# B&R Automation Studio project Parker_BMM_ST_V5_3147_V12 (part 11)

#### extrlift.c
```c
/********************************************************************
 * COPYRIGHT --  B&R China
 ********************************************************************
 * Program: extrlift
 * File: extrlift.c
 * Author: lijianjun
 * Created: March 06, 2013
 ********************************************************************
 * Implementation of program extrlift --- upward and downward
 ********************************************************************/

#include <bur/plctypes.h>

#ifdef _DEFAULT_INCLUDES
#include <AsDefault.h>
#endif

#define   INSTANCY_STOP_DECEL       3000

#define   INSTANCY_STOP_UP_DECEL    3000
#define   INSTANCY_STOP_DN_DECEL    3000
/**************************************************************************************
                            Function Declarations
**************************************************************************************/
void ExtrLiftTime( Mold_typ * pMold);
void ExtrLiftInverter( Mold_typ * pMold);
void ExtrLiftSwitch( Mold_typ * pMold);
void ExtrLiftDriveToggle_Drive(Mold_typ * pMold, ExtrLift_Fix_typ * pExtrLiftFix, ExtrLift_Para_typ * pExtrLiftPara);
REAL xTogLinearRTrans(REAL pTogLinPos);
/**************************************************************************************
     	        		I N I T U P  O F   T H E   T A S K
**************************************************************************************/
_INIT void init ( void )
{
	RTInfo_Task.enable = 1;
	RTInfo(&RTInfo_Task);

	tTask = RTInfo_Task.cycle_time/1000.0/1000.0;		/*  from us ---> s  */

	LMold.ExtrLift.Step = 30000;
	RMold.ExtrLift.Step = 30000;

	RMold.ExtrLift.vProfGen.Ts    = tTask;
	RMold.ExtrLift.vProfGen.accel = 800.0;
	RMold.ExtrLift.vProfGen.decel = 600.0;
	RMold.ExtrLift.vRamp.Ts       = tTask;
	RMold.ExtrLift.vRamp.Accel    = 1000;

	LMold.ExtrLift.vProfGen.Ts    = tTask;
	LMold.ExtrLift.vProfGen.accel = 800.0;
	LMold.ExtrLift.vProfGen.decel = 600.0;
	LMold.ExtrLift.vRamp.Ts       = tTask;
	LMold.ExtrLift.vRamp.Accel    = 1000;

	/* differentiator for evaluating the actual speed */
	vActHydDT2_L.Ts = tTask;	/* cycle time tTasks 			  */
	vActHydDT2_L.Tv = 1.0; 	/* derivative time constant [s]   */
	vActHydDT2_L.T1 = 5 * tTask; 	/* filter time constant 1 : 0.01s */
	vActHydDT2_L.T2 = 5 * tTask; 	/* filter time constant 2 : 0.01s */

	/* differentiator for evaluating the actual speed */
	vActHydDT2_R.Ts = tTask;	/* cycle time tTasks 			  */
	vActHydDT2_R.Tv = 1.0; 	/* derivative time constant [s]   */
	vActHydDT2_R.T1 = 5 * tTask; 	/* filter time constant 1 : 0.01s */
	vActHydDT2_R.T2 = 5 * tTask; 	/* filter time constant 2 : 0.01s */

	if( 10 > gMachineFix.ExtrLift.ToggleLinNodeNum ) gMachineFix.ExtrLift.ToggleLinNodeNum = 10;
	ToggleLinNodeNum = gMachineFix.ExtrLift.ToggleLinNodeNum;
	/* extrlift toggle linear */

	TogLinearR.enable = 1;
	TogLinearR.nNodes = ToggleLinNodeNum;
	TogLinearR.pNodes = &gMachineFix.ExtrLift.ToggleLin[0];

	xTogLinearR.enable = 1;
	xTogLinearR.nNodes = ToggleLinNodeNum;
	xTogLinearR.pNodes = &xToggleNodeR[0];

	memcpy(ToggleROld,gMachineFix.ExtrLift.ToggleLin,sizeof(gMachineFix.ExtrLift.ToggleLin));

} /* end of _INIT */

 /*************************************************************************************
        				C Y C L I C   P A R T   O F   T H E   T A S K
**************************************************************************************/

_CYCLIC void cyclic ( void )
{
	if(gMachinePara.ExtrLiftLower.accel < 20.0)gMachinePara.ExtrLiftLower.accel = 20.0;

	if(1 == gMachineIn.ExtrLiftInverterFault)
	{
		cntTime = cntTime + 1;
		if(cntTime >10000)cntTime =1000;
	}
	else
	{
		cntTime = 0;
	}

	if(cntTime > 100)
	{
		gAlarm.SwingInvertErr = 1;
	}

	/*--- 機構線性，強制線性化 ----*/
	if( ACTUATOR_ELECTRIC ==  gMachineFix.ExtrLift.eActuatorType)
	{
		int ToggleLinIndex;
		if( MECHANISM_LINEAR ==  gMachineFix.ExtrLift.eMechanismType )
		{
			bToggle_Init = 1;
			for(ToggleLinIndex = 1;ToggleLinIndex < (MAX_TOGGLE_LIN_NUM); ToggleLinIndex++)
			{
				int iSumR = 0;
				iSumR = gMachineFix.ExtrLift.Length / (ToggleLinNodeNum);
				gMachineFix.ExtrLift.ToggleLin[ToggleLinIndex].X = iSumR * ToggleLinIndex ;
				gMachineFix.ExtrLift.ToggleLin[ToggleLinIndex].Y = iSumR * ToggleLinIndex ;

				if( ToggleLinIndex >= ToggleLinNodeNum)
				{
					gMachineFix.ExtrLift.ToggleLin[ToggleLinIndex].X = gMachineFix.ExtrLift.Length ;
					gMachineFix.ExtrLift.ToggleLin[ToggleLinIndex].Y = gMachineFix.ExtrLift.Length ;
				}

			}
		}
		else if( MECHANISM_TOGGLE ==  gMachineFix.ExtrLift.eMechanismType  )
		{
			if(1 == bToggle_Init)
			{
				bToggle_Init = 0;

				// clear ToggleLin table
				for(ToggleLinIndex = 1;ToggleLinIndex < (MAX_TOGGLE_LIN_NUM); ToggleLinIndex++)
				{

					if(ToggleLinIndex <ToggleLinNodeNum )
					{
						gMachineFix.ExtrLift.ToggleLin[ToggleLinIndex].X = 0 ;
						gMachineFix.ExtrLift.ToggleLin[ToggleLinIndex].Y = 0 ;
					}
					else
					{
						gMachineFix.ExtrLift.ToggleLin[ToggleLinIndex].X = gMachineFix.ExtrLift.Length ;
						gMachineFix.ExtrLift.ToggleLin[ToggleLinIndex].Y = gMachineFix.ExtrLift.Length ;
					}
				}

			}
		}
	}

	int i;
	for(i=0;i<MAX_TOGGLE_LIN_NUM;i++)
	{
		xToggleNodeR[i].X = gMachineFix.ExtrLift.ToggleLin[i].Y;
		xToggleNodeR[i].Y = gMachineFix.ExtrLift.ToggleLin[i].X;
	}

	if( 10 > gMachineFix.ExtrLift.ToggleLinNodeNum ) gMachineFix.ExtrLift.ToggleLinNodeNum = 10;
	else if( 30 < gMachineFix.ExtrLift.ToggleLinNodeNum ) gMachineFix.ExtrLift.ToggleLinNodeNum = 30;
	ToggleLinNodeNum = gMachineFix.ExtrLift.ToggleLinNodeNum;
	//TogLinear  update

	if(memcmp(ToggleROld,gMachineFix.ExtrLift.ToggleLin,sizeof(gMachineFix.ExtrLift.ToggleLin)) != 0
		|| oldToggleLinNodeNum != ToggleLinNodeNum)
	{
		TogLinearR.update = 1;
		TogLinearR.nNodes = ToggleLinNodeNum;
		memcpy(ToggleROld,gMachineFix.ExtrLift.ToggleLin,sizeof(gMachineFix.ExtrLift.ToggleLin));

		xTogLinearR.update = 1;
		xTogLinearR.nNodes = ToggleLinNodeNum;
		HydLinear(&xTogLinearR);
	}

	oldToggleLinNodeNum = ToggleLinNodeNum;

	/*  ExtruderLift Up & Dn limit   */
	RMold.TransDIn.ExtruderLiftUpLimit = gMachineIn.ExtruderLiftUpLimit;
	LMold.TransDIn.ExtruderLiftUpLimit = gMachineIn.ExtruderLiftUpLimit;

	RMold.TransDIn.ExtruderLiftDnLimit = gMachineIn.ExtruderLiftDnLimit;
	LMold.TransDIn.ExtruderLiftDnLimit = gMachineIn.ExtruderLiftDnLimit;

	/*  valve output*/
	gMachineOut.ExtrLiftUp 		= (LMold.ValveOut.ExtrLiftUp| RMold.ValveOut.ExtrLiftUp);
	gMachineOut.ExtrLiftUpCheck = (LMold.ValveOut.ExtrLiftUpCheck| RMold.ValveOut.ExtrLiftUpCheck);  /* 上止回閥*/
	if(1 == gMachineFix.Option.bExtrLiftUpFastValve)
	{
		gMachineOut.ExtrLiftUpFast  = (LMold.ValveOut.ExtrLiftUpFast | RMold.ValveOut.ExtrLiftUpFast);	 /* 上快速閥*/
	}
	gMachineOut.ExtrLiftDn 		= (LMold.ValveOut.ExtrLiftDn | RMold.ValveOut.ExtrLiftDn);

	/* velocity  */

	if(ACTUATOR_HYD == gMachineFix.ExtrLift.eActuatorType)
	{
		vActHydDT2_R.u = RMold.ExtrLift.mmAs;
	}
	else if(ACTUATOR_ELECTRIC == gMachineFix.ExtrLift.eActuatorType)
	{
		if(TogLinearR.status != 0)  //LinNotOK
		{
			vActHydDT2_R.u = RMold.ExtrLift.mmAs;
		}
		else
		{
			vActHydDT2_R.u = RMold.ExtrLift.mmAsDrive;
		}
	}

	HydDT2(&vActHydDT2_R);
	RMold.ExtrLift.v_act = vActHydDT2_R.y;

	/*  run function  */
	if(ACTUATOR_HYD == gMachineFix.ExtrLift.eActuatorType) //Hydraulic
	{
		if(0 == gMachineFix.Option.bHideLeftStation)  // two mold
		{
			ExtrLiftSwitch(&LMold);
		}
		ExtrLiftSwitch(&RMold);
	}
	else if(ACTUATOR_ELECTRIC == gMachineFix.ExtrLift.eActuatorType) //Electric
	{
		//		if(0 == gMachineFix.Option.bHideLeftStation)  // two mold
		//		{
		//			ExtrLiftDriveToggle_Drive(&LMold, &gMachineFix.ExtrLift, &gMachinePara.Extrlift);
		//		}
		ExtrLiftDriveToggle_Drive(&RMold, &gMachineFix.ExtrLift, &gMachinePara.Extrlift);
	}

	/*------------- ActuatorType--------------- */
	gMachineFix.ExtrLift.eActuatorType;

	/*------------ PressueOutputType--------------- */
	gMachineFix.ExtrLift.ePressueOutputType;

	/*------------ FluxOutputType--------------- */
	gMachineFix.ExtrLift.eFluxOutputType;

	/*---------------Motor Trand-------------*/
	gMotorTrace.Extrlift.Position 		= RMold.ExtrLift.mmAs;

} /* end of _CYCLIC */

void ExtrLiftTime( Mold_typ * pMold)
{

	/* ------------------ Step Machine Control ------------------ */
	switch ( pMold->ExtrLift.Step )
	{
		/*------------------ stop all the output ------------------*/
		case 0:
			pMold->ValveOut.ExtrLiftUp  = 0;
			pMold->ActInfo.ExtrLiftUp = 0;
			pMold->ActInfo.ExtrLiftDn = 0;

			pMold->ExtrLift.Timer.IN = 0;
			break;

		/*------------------ Extr Lift -------------------- */
		case 100: 	/* ExtrLift delay*/

			if(pMold->TimeSet.ExtrLiftUpDelay != 0)
			{
				pMold->ExtrLift.Timer.IN = 1;
				pMold->ExtrLift.Timer.PT = pMold->TimeSet.ExtrLiftUpDelay;
				pMold->ExtrLift.Step 	= 200;
			}
			else
			{
				pMold->ExtrLift.Step = 300;
			}
			break;

		case 200: 	/* delay ok */
			pMold->TimeDis.ExtrLiftUpDelay = pMold->ExtrLift.Timer.ET;
			if (1 == pMold->ExtrLift.Timer.Q)
			{
				pMold->ExtrLift.Timer.IN     = 0;
				//				pMold->TimeDis.ExtrLiftUpDelay = 0;
				pMold->ExtrLift.Step = 300;
			}
			break;

		case 300:
			if(pMold->TimeSet.ExtrLiftUpHoldTime != 0)
			{
				pMold->ExtrLift.Timer.IN = 1;
				pMold->ExtrLift.Timer.PT = pMold->TimeSet.ExtrLiftUpHoldTime;
				pMold->ExtrLift.Step = 400;
			}
			else
			{
				pMold->ExtrLift.Step = 2900;
			}
			break;

		case 400:
			pMold->ActInfo.ExtrLiftUp = 1;
			pMold->ActInfo.ExtrLiftDn = 0;
			pMold->ValveOut.ExtrLiftUp       = 1;

			pMold->TimeDis.ExtrLiftUpHoldTime = pMold->ExtrLift.Timer.ET;
			if (1 == pMold->ExtrLift.Timer.Q)
			{
				pMold->ValveOut.ExtrLiftUp     = 0;
				pMold->ExtrLift.Timer.IN = 0;
				//				pMold->TimeDis.ExtrLiftUpHoldTime = 0;
				pMold->ExtrLift.Step = 500;
			}
			break;

		case 500:
			pMold->ActInfo.ExtrLiftUp = 0;
			pMold->ActInfo.ExtrLiftDn = 0;/*Test*/
			pMold->ValveOut.ExtrLiftUp       = 0;

			pMold->ExtrLift.Step = 2900;
			break;

		case 2900:
			pMold->ExtrLift.Timer.IN    = 0;

			pMold->TimeDis.ExtrLiftUpDelay = 0;
			pMold->TimeDis.ExtrLiftUpHoldTime = 0;
			pMold->TimeDis.ExtrLiftSlowTime = 0;

			pMold->ActInfo.ExtrLiftUp = 0;
			pMold->ActInfo.ExtrLiftDn = 0;
			pMold->ValveOut.ExtrLiftUp       = 0;

			pMold->ExtrLift.Step = 3000;
			break;
		case 3000:
			break;

		case 5000:					/*  Manual up */

			pMold->ActInfo.ExtrLiftUp = 1;
			pMold->ActInfo.ExtrLiftDn = 0;

			if((0 == pMold->TransDIn.ExtruderLiftUpLimit) && (0 == pMold->TransDIn.ExtruderLiftDnLimit))
			{
				pMold->ValveOut.ExtrLiftUp       = 0;
			}
			else
			{
				if(1 == pMold->TransDIn.ExtruderLiftUpLimit)
				{
					pMold->ValveOut.ExtrLiftUp       = 0;
				}
				else
				{
					pMold->ValveOut.ExtrLiftUp       = 1;
				}
			}
			break;

		case 15000:					/*  Manual down */
			pMold->ActInfo.ExtrLiftUp = 0;
			pMold->ActInfo.ExtrLiftDn = 0;
			pMold->ValveOut.ExtrLiftUp       = 0;

			break;

		/*--------------- Manual action stop -----------------*/
		case 20000:
			pMold->ExtrLift.Timer.IN = 0;

			pMold->ActInfo.ExtrLiftUp = 0;
			pMold->ActInfo.ExtrLiftDn = 0;
			pMold->ValveOut.ExtrLiftUp       = 0;

			pMold->ExtrLift.Step = 0;
			break;

		/*--------------- Instance stop -----------------*/
		case 30000:
			pMold->ExtrLift.Timer.IN = 0;

			pMold->ActInfo.ExtrLiftUp = 0;
			pMold->ActInfo.ExtrLiftDn = 0;
			pMold->ValveOut.ExtrLiftUp       = 0;

			pMold->ExtrLift.Step = 0;
			break;

		/*--------------- error -----------------*/
		case 40000:
			pMold->ExtrLift.Timer.IN  = 0;
			pMold->ActInfo.ExtrLiftUp = 0;
			pMold->ActInfo.ExtrLiftDn = 0;
			pMold->ValveOut.ExtrLiftUp       = 0;

			pMold->ExtrLift.Step = 0;
			break;
	}/* end of switch */
}/*end of function */

void ExtrLiftInverter( Mold_typ * pMold)
{
	if(0 == pMold->TimeSet.ExtrLiftSlowTime)pMold->TimeSet.ExtrLiftSlowTime = 1000;

	switch ( pMold->ExtrLift.Step)
	{
		/*------------------ stop all the output ------------------*/
		case 0:
			pMold->ValveOut.ExtrLiftUp   = 0;
			pMold->ExtrLift.v_set = 0.0;

			pMold->ActInfo.ExtrLiftUp = 0;
			pMold->ActInfo.ExtrLiftDn = 0;

			pMold->ExtrLift.Timer.IN = 0;
			break;

		/*------------------ Extr Lift -------------------- */
		case 100: 	/* ExtrLift delay*/
			if(pMold->TimeSet.ExtrLiftUpDelay != 0)
			{
				pMold->ExtrLift.Timer.IN = 1;
				pMold->ExtrLift.Timer.PT = pMold->TimeSet.ExtrLiftUpDelay;
				pMold->ExtrLift.Step 	= 200;
			}
			else
			{
				pMold->ExtrLift.Step = 300;
			}
			break;

		case 200: 	/* delay ok */
			pMold->TimeDis.ExtrLiftUpDelay = pMold->ExtrLift.Timer.ET;
			if (1 == pMold->ExtrLift.Timer.Q)
			{
				pMold->ExtrLift.Timer.IN     = 0;
				pMold->TimeDis.ExtrLiftUpDelay = 0;
				pMold->ExtrLift.Step = 300;
			}
			break;

		case 300:
			pMold->ExtrLift.Timer.IN = 1;
			pMold->ExtrLift.Timer.PT = pMold->TimeSet.ExtrLiftSlowTime;

			pMold->ExtrLift.vRamp.Internal.Once = 0;
			pMold->ExtrLift.vRamp.Set = 0.0;

			pMold->ExtrLift.vRamp.Ts = 0.002;
			pMold->ExtrLift.vRamp.Accel = gMachinePara.ExtrLiftLower.accel;
			if(pMold->ExtrLift.vRamp.Accel < 10)pMold->ExtrLift.vRamp.Accel = 100;

			HydSCurveRamp(&pMold->ExtrLift.vRamp);
			pMold->ExtrLift.v_set = pMold->ExtrLift.vRamp.Out;

			pMold->ExtrLift.Step = 400;
			break;

		case 400:
			pMold->ActInfo.ExtrLiftUp = 1;
			pMold->ActInfo.ExtrLiftDn = 0;
			pMold->ValveOut.ExtrLiftUp       = 1;

			pMold->ExtrLift.vRamp.Set = gMachinePara.ExtrLiftLower.vLowerQuick;
			HydSCurveRamp(&pMold->ExtrLift.vRamp);
			pMold->ExtrLift.v_set = pMold->ExtrLift.vRamp.Out;

			pMold->TimeDis.ExtrLiftUpHoldTime = pMold->ExtrLift.Timer.ET;
			if(1 == gMachineIn.ExtrLowerSlowLimit || pMold->TimeDis.ExtrLiftUpHoldTime >= pMold->TimeSet.ExtrLiftUpHoldTime )
			{
				pMold->ExtrLift.Step = 500;
			}

			pMold->TimeDis.ExtrLiftSlowTime = pMold->ExtrLift.Timer.ET;
			if (1 == pMold->ExtrLift.Timer.Q)
			{
				pMold->ExtrLift.v_set = 0.0;
				pMold->ValveOut.ExtrLiftUp      = 0;
				pMold->ExtrLift.Timer.IN = 0;
				pMold->ExtrLift.Step = 40000;
			}
			break;

		case 500:
			pMold->ValveOut.ExtrLiftUp = 1;

			pMold->ExtrLift.vRamp.Set = gMachinePara.ExtrLiftLower.vLowerSlow;
			HydSCurveRamp(&pMold->ExtrLift.vRamp);
			pMold->ExtrLift.v_set = pMold->ExtrLift.vRamp.Out;

			pMold->TimeDis.ExtrLiftSlowTime = pMold->ExtrLift.Timer.ET;
			if (1 == pMold->ExtrLift.Timer.Q)
			{
				pMold->ExtrLift.v_set = 0.0;
				pMold->ValveOut.ExtrLiftUp      = 0;
				pMold->ExtrLift.Timer.IN = 0;
				pMold->ExtrLift.Step = 40000;
			}

			if(1 == gMachineIn.ExtrLowerLimit)
			{
				pMold->ExtrLift.Timer.IN = 0;
				pMold->ExtrLift.Step = 600;
			}
			break;

		case 600:
			pMold->ExtrLift.vRamp.Accel = 1600;
			pMold->ExtrLift.vRamp.Set = 0.0;
			HydSCurveRamp(&pMold->ExtrLift.vRamp);
			pMold->ExtrLift.v_set = pMold->ExtrLift.vRamp.Out;

			if(pMold->ExtrLift.v_set < 0.1 && pMold->ExtrLift.v_set > -0.1)
			{
				pMold->ExtrLift.v_set = 0.0;
				pMold->ExtrLift.Step = 700;
			}
			break;

		case 700:
			pMold->ActInfo.ExtrLiftUp = 0;
			pMold->ActInfo.ExtrLiftDn = 0;
			pMold->ValveOut.ExtrLiftUp       = 0;
			pMold->ExtrLift.v_set     = 0.0;

			pMold->ExtrLift.Step = 2900;
			break;

		case 2900:
			pMold->ExtrLift.Timer.IN    = 0;

			pMold->TimeDis.ExtrLiftUpDelay = 0;

			pMold->ActInfo.ExtrLiftUp = 0;
			pMold->ActInfo.ExtrLiftDn = 0;
			pMold->ValveOut.ExtrLiftUp       = 0;
			pMold->ExtrLift.v_set     = 0.0;

			pMold->ExtrLift.Step = 3000;
			break;
		case 3000:
			break;

		case 5000:					/*  Manual up */
			pMold->ActInfo.ExtrLiftUp = 1;
			pMold->ActInfo.ExtrLiftDn = 0;
			pMold->ValveOut.ExtrLiftUp       = 1;

			pMold->ExtrLift.v_set = gMachinePara.ExtrLiftLower.vLowerSlow;
			break;

		case 15000:					/*  Manual down */
			pMold->ActInfo.ExtrLiftUp = 0;
			pMold->ActInfo.ExtrLiftDn = 0;
			pMold->ValveOut.ExtrLiftUp       = 0;
			break;

		/*--------------- Manual action stop -----------------*/
		case 20000:
			pMold->ExtrLift.Timer.IN = 0;

			pMold->ActInfo.ExtrLiftUp = 0;
			pMold->ActInfo.ExtrLiftDn = 0;
			pMold->ValveOut.ExtrLiftUp       = 0;

			pMold->ExtrLift.vRamp.Internal.Once = 0;
			pMold->ExtrLift.vRamp.Set = pMold->ExtrLift.v_set;

			pMold->ExtrLift.vRamp.Ts = 0.002;
			pMold->ExtrLift.vRamp.Accel = gMachinePara.ExtrLiftLower.accel;
			if(pMold->ExtrLift.vRamp.Accel < 10)pMold->ExtrLift.vRamp.Accel = 100;

			HydSCurveRamp(&pMold->ExtrLift.vRamp);
			pMold->ExtrLift.v_set = pMold->ExtrLift.vRamp.Out;

			pMold->ExtrLift.Step = 21000;
			break;

		case 21000:
			pMold->ExtrLift.vRamp.Accel = 2000;
			pMold->ExtrLift.vRamp.Set = 0.0;
			HydSCurveRamp(&pMold->ExtrLift.vRamp);
			pMold->ExtrLift.v_set = pMold->ExtrLift.vRamp.Out;

			if(pMold->ExtrLift.v_set < 0.1 && pMold->ExtrLift.v_set > -0.1)
			{
				pMold->ExtrLift.v_set = 0.0;
				pMold->ExtrLift.Step = 0;
			}
			break;

		/*--------------- Instance stop -----------------*/
		case 30000:
			pMold->ExtrLift.Timer.IN = 0;

			pMold->ActInfo.ExtrLiftUp = 0;
			pMold->ActInfo.ExtrLiftDn = 0;
			pMold->ValveOut.ExtrLiftUp   = 0;
			pMold->ExtrLift.v_set = 0.0;

			pMold->ExtrLift.Step = 0;
			break;

		/*--------------- error -----------------*/
		case 40000:
			pMold->ExtrLift.Timer.IN  = 0;
			pMold->ActInfo.ExtrLiftUp = 0;
			pMold->ActInfo.ExtrLiftDn = 0;
			pMold->ValveOut.ExtrLiftUp   = 0;
			pMold->ExtrLift.v_set = 0.0;

			pMold->ExtrLift.Step = 0;
			break;
	}/* end of switch */

}/*end of function */

void ExtrLiftSwitch( Mold_typ * pMold)
{
	switch ( pMold->ExtrLift.Step )
	{
		/*------------------ stop all the output ------------------*/
		case 0:
			pMold->ActInfo.ExtrLiftUp = 0;
			pMold->ActInfo.ExtrLiftDn = 0;
			pMold->ValveOut.ExtrLiftUp     = 0;
			pMold->ValveOut.ExtrLiftUpCheck    = 0;
			pMold->ValveOut.ExtrLiftUpFast     = 0;
			pMold->ValveOut.ExtrLiftDn 	 = 0;

			pMold->ExtrLift.Timer.IN = 0;
			pMold->ExtrLift.LimitTimer.IN = 0; //ipis0219
			break;

		/*------------------ Extr Lift up-------------------- */
		case 100: 	/* ExtrLift delay*/
			if(pMold->Option.ExtrLift)
			{
				if(pMold->TimeSet.ExtrLiftUpDelay != 0)
				{
					pMold->ExtrLift.Timer.IN = 1;
					pMold->ExtrLift.Timer.PT = pMold->TimeSet.ExtrLiftUpDelay;
					pMold->ExtrLift.Step 	= 200;
				}
				else
				{
					pMold->ExtrLift.Step = 300;
				}
			}
			else
			{
				pMold->ExtrLift.Step = 2900;
			}
			break;

		case 200: 	/* delay ok */
			pMold->TimeDis.ExtrLiftUpDelay = pMold->ExtrLift.Timer.ET;
			if (1 == pMold->ExtrLift.Timer.Q)
			{
				pMold->ExtrLift.Timer.IN     = 0;
				//	pMold->TimeDis.ExtrLiftUpDelay = 0;

				pMold->ExtrLift.Step = 300;
			}
			break;

		case 300:
			if (0 == pMold->TransDIn.ExtruderLiftUpLimit)
			{
				pMold->ExtrLift.LimitTimer.IN = 1; //ipis0219
				pMold->ExtrLift.LimitTimer.PT = pMold->TimeSet.ExtrLiftUpAlarmTime; //ipis0219

				pMold->ExtrLift.Step = 400;
			}
			else
			{
				pMold->ExtrLift.Step = 500;
			}
			break;

		case 400:
			pMold->ActInfo.ExtrLiftUp = 1;
			pMold->ActInfo.ExtrLiftDn = 0;
			pMold->ValveOut.ExtrLiftUp   = 1;
			pMold->ValveOut.ExtrLiftUpCheck    = 0;
			pMold->ValveOut.ExtrLiftUpFast     = 1;
			pMold->ValveOut.ExtrLiftDn 	 = 0;

			pMold->TimeDis.ExtrLiftUpAlarmTime = pMold->ExtrLift.LimitTimer.ET;

			if (1 == pMold->TransDIn.ExtruderLiftUpLimit)
			{

				if(pMold->TimeSet.ExtrLiftUpHoldTime != 0)
				{
					pMold->ExtrLift.Timer.IN = 1;
					pMold->ExtrLift.Timer.PT = pMold->TimeSet.ExtrLiftUpHoldTime;
					pMold->ExtrLift.Step = 450;
				}
				else
				{
					pMold->ExtrLift.Step = 500;
				}
			}
			break;
		case 450:
			pMold->ValveOut.ExtrLiftUpFast     = 0;

			pMold->TimeDis.ExtrLiftUpHoldTime = pMold->ExtrLift.Timer.ET;
			if (1 == pMold->ExtrLift.Timer.Q)
			{
				pMold->ValveOut.ExtrLiftUp      = 0;
				pMold->ExtrLift.Timer.IN = 0;

				pMold->ExtrLift.Step = 500;
			}

			break;

		case 500:
			pMold->ActInfo.ExtrLiftUp = 0;
			pMold->ActInfo.ExtrLiftDn = 0;
			pMold->ValveOut.ExtrLiftUp      = 0;
			pMold->ValveOut.ExtrLiftUpCheck    = 0;
			pMold->ValveOut.ExtrLiftUpFast     = 0;
			pMold->ValveOut.ExtrLiftDn 	  = 0;

			pMold->ExtrLift.LimitTimer.IN = 0;
			if (1 == gMachineInfo.Auto)
			{
				pMold->ExtrLift.Step = 10100;
			}
			else
			{
				pMold->ExtrLift.Step = 2900;
			}

			break;

		case 2900:
			pMold->ExtrLift.Timer.IN    = 0;
			pMold->ExtrLift.LimitTimer.IN = 0;

			//			//gExSPC
			//			if(pMold == & LMold)
			//			{
			//				gExSPC[ExIndex].LMold.tExtrLift = pMold->ExtrLift.LimitTimer.ET/100.0;
			//			}
			//			else
			//			{
			//				gExSPC[ExIndex].RMold.tExtrLift = pMold->ExtrLift.LimitTimer.ET/100.0;
			//			}

			//	pMold->TimeDis.ExtrLiftUpDelay = 0;
			//	pMold->TimeDis.ExtrLiftUpHoldTime = 0;
			//	pMold->TimeDis.ExtrLiftDnHoldTime = 0;

			//	pMold->TimeDis.ExtrLiftUpHoldTime = 0;
			//	pMold->TimeDis.ExtrLiftDnHoldTime = 0;

			pMold->ActInfo.ExtrLiftUp = 0;
			pMold->ActInfo.ExtrLiftDn = 0;
			pMold->ValveOut.ExtrLiftUp      = 0;
			pMold->ValveOut.ExtrLiftUpCheck = 0;
			pMold->ValveOut.ExtrLiftUpFast  = 0;
			pMold->ValveOut.ExtrLiftDn 	  = 0;

			pMold->ExtrLift.Step = 3000;
			break;

		case 3000:
			break;

		case 5000:					/*  Manual up */
			pMold->ActInfo.ExtrLiftUp = 1;
			pMold->ActInfo.ExtrLiftDn = 0;

			pMold->ValveOut.ExtrLiftUp    = 1;
			pMold->ValveOut.ExtrLiftUpCheck  = 0;
			pMold->ValveOut.ExtrLiftUpFast   = 0;
			pMold->ValveOut.ExtrLiftDn 	  = 0;

			break;

		/*------------------ Extr Lift down -------------------- */
		case 10100:
			if (pMold->TimeSet.ExtrLiftDnDelay != 0)
			{
				pMold->ExtrLift.Timer.IN = 1;
				pMold->ExtrLift.Timer.PT = pMold->TimeSet.ExtrLiftDnDelay;
				pMold->ExtrLift.Step = 10200;
			}
			else
			{
				pMold->ExtrLift.Step = 10300;
			}
			break;
		case 10200:
			pMold->TimeDis.ExtrLiftDnDelay = pMold->ExtrLift.Timer.ET;
			if (1 == pMold->ExtrLift.Timer.Q)
			{
				pMold->ExtrLift.Timer.IN = 0;
				//	pMold->TimeDis.ExtrLiftDnDelay = 0;
				pMold->ExtrLift.Step = 10300;
			}
			break;
		case 10300:
			if ( 0 == gMachineIn.ExtruderLiftDnLimit)
			{
				pMold->ExtrLift.LimitTimer.IN = 1;
				pMold->ExtrLift.LimitTimer.PT = pMold->TimeSet.ExtrLiftDnAlarmTime;

				pMold->ExtrLift.Step = 10400;
			}
			else
			{
				pMold->ExtrLift.Step = 10500;
			}
			break;
		case 10400:
			pMold->ActInfo.ExtrLiftUp = 0;
			pMold->ActInfo.ExtrLiftDn = 1;
			pMold->ValveOut.ExtrLiftUp  	= 0;
			pMold->ValveOut.ExtrLiftUpCheck = 1;
			pMold->ValveOut.ExtrLiftUpFast  = 0;
			pMold->ValveOut.ExtrLiftDn 	    = 1;

			pMold->TimeDis.ExtrLiftDnAlarmTime = pMold->ExtrLift.LimitTimer.ET;

			if ( 1 == gMachineIn.ExtruderLiftDnLimit)
			{
				if(pMold->TimeSet.ExtrLiftDnHoldTime != 0)
				{
					pMold->ExtrLift.Timer.IN = 1;
					pMold->ExtrLift.Timer.PT = pMold->TimeSet.ExtrLiftDnHoldTime;
					pMold->ExtrLift.Step = 10450;
				}
				else
				{
					pMold->ExtrLift.Step = 10500;
				}
			}
			break;
		case 10450:
			pMold->TimeDis.ExtrLiftDnHoldTime = pMold->ExtrLift.Timer.ET;
			if (1 == pMold->ExtrLift.Timer.Q)
			{
				pMold->ValveOut.ExtrLiftUp    = 0;
				pMold->ValveOut.ExtrLiftUpCheck = 0;
				pMold->ValveOut.ExtrLiftUpFast  = 0;
				pMold->ValveOut.ExtrLiftDn 	  = 0;
				pMold->ExtrLift.Timer.IN = 0;
				//				pMold->TimeDis.ExtrLiftDnHoldTime = 0;
				pMold->ExtrLift.Step = 10500;
			}
			break;
		case 10500:
			pMold->ActInfo.ExtrLiftUp = 0;
			pMold->ActInfo.ExtrLiftDn = 0;
			pMold->ValveOut.ExtrLiftUp      = 0;
			pMold->ValveOut.ExtrLiftUpCheck = 0;
			pMold->ValveOut.ExtrLiftUpFast  = 0;
			pMold->ValveOut.ExtrLiftDn 	  = 0;
			pMold->ExtrLift.Timer.IN    = 0;
			pMold->ExtrLift.LimitTimer.IN = 0;

			pMold->ExtrLift.Step 	  = 13000;
			break;

		case 13000:

			break;

		case 15000:					/*  Manual down */
			pMold->ActInfo.ExtrLiftUp = 0;
			pMold->ActInfo.ExtrLiftDn = 1;
			pMold->ValveOut.ExtrLiftUp    = 0;
			pMold->ValveOut.ExtrLiftUpCheck  = 1;
			pMold->ValveOut.ExtrLiftUpFast   = 0;
			pMold->ValveOut.ExtrLiftDn 	  = 1;

			break;

		/*--------------- Manual action stop -----------------*/
		case 20000:
			pMold->ExtrLift.Timer.IN = 0;

			pMold->ActInfo.ExtrLiftUp = 0;
			pMold->ActInfo.ExtrLiftDn = 0;
			pMold->ValveOut.ExtrLiftUp       = 0;
			pMold->ValveOut.ExtrLiftUpFast 	 = 0;

			pMold->ValveOut.ExtrLiftUpCheck = 0;
			pMold->ValveOut.ExtrLiftDn 	  	= 0;

			pMold->ExtrLift.Step = 0;
			break;

		/*--------------- Instance stop -----------------*/
		case 30000:
			pMold->ExtrLift.Timer.IN = 0;

			pMold->ActInfo.ExtrLiftUp = 0;
			pMold->ActInfo.ExtrLiftDn = 0;
			pMold->ValveOut.ExtrLiftUp       = 0;
			pMold->ValveOut.ExtrLiftUpFast 	 = 0;

			pMold->ValveOut.ExtrLiftUpCheck = 0;
			pMold->ValveOut.ExtrLiftDn 	  	= 0;

			pMold->ExtrLift.Step = 0;
			break;

		/*--------------- error -----------------*/
		case 40000:
			pMold->ExtrLift.Timer.IN  = 0;

			pMold->ActInfo.ExtrLiftUp = 0;
			pMold->ActInfo.ExtrLiftDn = 0;
			pMold->ValveOut.ExtrLiftUp       = 0;
			pMold->ValveOut.ExtrLiftUpFast 	 = 0;

			pMold->ValveOut.ExtrLiftUpCheck = 0;
			pMold->ValveOut.ExtrLiftDn 	  	= 0;

			pMold->ExtrLift.Step = 0;
			break;
	}/* end of switch */

	/* ----------------- ExtrLift Up / down timeout --------------------  */
	if(1 == pMold->ExtrLift.LimitTimer.Q && 1 == gMachineInfo.TimeLimit)
	{
		if(pMold->ExtrLift.Step < 500 && pMold->ExtrLift.Step > 200)		/* ExtrLift Up  */
		{
			pMold->Alarm.ExtrLiftNotAtUpPos = 1;
		}

		if(pMold->ExtrLift.Step < 10500 && pMold->ExtrLift.Step > 10200)		/* ExtrLift Dn  */
		{
			pMold->Alarm.ExtrLiftNotAtDnPos = 1;
		}

		pMold->ExtrLift.LimitTimer.IN = 0;
		pMold->ExtrLift.Step = 40000;

		if(gMachineInfo.Auto)
		{
			gMachineInfo.ExtrliftAlarmReqSemiAutoFlag = 1;
		}
	}
}

void ExtrLiftDriveToggle_Drive(Mold_typ * pMold, ExtrLift_Fix_typ * pExtrLiftFix, ExtrLift_Para_typ * pExtrLiftPara)
{
	if(pMold == & LMold)
	{
		pExtrLiftFix->pMax = 100;
	}
	else
	{
		pExtrLiftFix->pMax = 100;
	}

	if(1 == gMachineOut.OilPump)
	{
		if(tErrorDelay >= tTask)tErrorDelay = tErrorDelay - tTask;
		if(tErrorDelay < tTask)
		{
			if(pMold == & LMold)
			{
				LMold.HwAlarm.ExtrLiftNetworkErr = !LMold.ExtrLift.NetworkInit;
				LMold.HwAlarm.ExtrLiftPowerOn    = !LMold.ExtrLift.PowerOn;
			}
			else
			{
				RMold.HwAlarm.ExtrLiftNetworkErr = !RMold.ExtrLift.NetworkInit;
				RMold.HwAlarm.ExtrLiftPowerOn    = !RMold.ExtrLift.PowerOn;
			}
		}

		if((RMold.HwAlarm.ExtrLiftNetworkErr ||RMold.HwAlarm.ExtrLiftPowerOn)/*||(LMold.HwAlarm.ExtrLiftNetworkErr ||LMold.HwAlarm.ExtrLiftPowerOn)*/)
		{
			gMachineOut.OilPump = 0;
			gPROCESS_info.oilpumpStop = 1;   //request manual mode
		}
	}
	else
	{
		tErrorDelay = 0.5;
		//		if(pMold == & LMold)
		//		{
		////			LMold.HwAlarm.ExtrLiftNetworkErr = 0;
		////			LMold.HwAlarm.ExtrLiftPowerOn    = 0;
		//		}
		//		else
		//		{
		////			RMold.HwAlarm.ExtrLiftNetworkErr = 0;
		////			RMold.HwAlarm.ExtrLiftPowerOn    = 0;
		//		}
	}

	/* ------------- extrLift axis alarms ------------- */

	pMold->HwAlarm.ExtrLiftAxisErr    = RMold.ExtrLift.Error;

	 /*********************************************************************************
  	**                            HMI data value to PLC                             **
  	*********************************************************************************/
	if(pExtrLiftFix->Length < 10.0)pExtrLiftFix->Length = 60.0;
	if(pExtrLiftFix->Tolerance < 0.1)pExtrLiftFix->Tolerance = 2.0;
	pMold->ExtrLift.Tolerance = pExtrLiftFix->Tolerance;

	if(pExtrLiftFix->Up.V_Max < 30.0)pExtrLiftFix->Up.V_Max = 1000.0;
	if(pExtrLiftFix->Dn.V_Max < 30.0)pExtrLiftFix->Dn.V_Max = 1000.0;

	if(pExtrLiftFix->Up.VoltageMax > -3.0)pExtrLiftFix->Up.VoltageMax = -10.0;
	if(pExtrLiftFix->Dn.VoltageMax < 3.0 )pExtrLiftFix->Dn.VoltageMax = 10.0;

	pMold->ExtrLift.S_Up = pExtrLiftPara->S_Up;
	pMold->ExtrLift.V_Up = pExtrLiftPara->V_Up * pExtrLiftFix->Up.V_Max/100.0;

	pMold->ExtrLift.S_Dn = pExtrLiftPara->S_Dn;
	pMold->ExtrLift.V_Dn = pExtrLiftPara->V_Dn * pExtrLiftFix->Dn.V_Max/100.0;

	if(0 == pExtrLiftPara->V_DnReset)pExtrLiftPara->V_DnReset = 2.0;
	pMold->ExtrLift.V_DnReset = pExtrLiftPara->V_DnReset * pExtrLiftFix->Dn.V_Max/100.0;

	if(pExtrLiftFix->Up.accel_stop < 100)pExtrLiftFix->Up.accel_stop = INSTANCY_STOP_UP_DECEL;
	if(pExtrLiftFix->Dn.accel_stop < 100)pExtrLiftFix->Dn.accel_stop = INSTANCY_STOP_DN_DECEL;
    /*********************************************************************************
   **                            linear calibration status                        **
   *********************************************************************************/
   /* get calibration data  */
	if(pExtrLiftFix->Max < pExtrLiftFix->Zero)
	{
		pMold->ExtrLift.ZeroPos = pExtrLiftFix->Max;
		pMold->ExtrLift.MaxPos  = pExtrLiftFix->Zero;
	}
	else
	{
		pMold->ExtrLift.MaxPos  = pExtrLiftFix->Max;
		pMold->ExtrLift.ZeroPos = pExtrLiftFix->Zero;
	}

	if(pMold->ExtrLift.ZeroPos != 0            						&&
		pMold->ExtrLift.MaxPos > (pMold->ExtrLift.ZeroPos + 3000)  	&&
		pMold->ExtrLift.As     > (pMold->ExtrLift.ZeroPos - 1000)   &&
		pMold->ExtrLift.As     < (RMold.ExtrLift.MaxPos  + 5000))
	{
		pMold->ExtrLift.CalOK = pMold->ExtrLift.NetworkInit;
	}
	else
	{
		pMold->ExtrLift.CalOK = 0;
	}

	pExtrLiftFix->CalibOK = pMold->ExtrLift.CalOK;

	if(1 == pMold->ExtrLift.CalOK)
	{
		if(pExtrLiftFix->Max < pExtrLiftFix->Zero)
		{
			pMold->ExtrLift.mmAsDrive = 1.0 *(pMold->ExtrLift.MaxPos - pMold->ExtrLift.As) * pExtrLiftFix->Length /
				(pMold->ExtrLift.MaxPos - pMold->ExtrLift.ZeroPos);
		}
		else
		{
			pMold->ExtrLift.mmAsDrive = 1.0 *(pMold->ExtrLift.As - pMold->ExtrLift.ZeroPos) * pExtrLiftFix->Length /
				(pMold->ExtrLift.MaxPos - pMold->ExtrLift.ZeroPos);
		}
	}
	else
	{
		pMold->ExtrLift.mmAsDrive = pMold->ExtrLift.mmAsDrive;
		//		pMold->ExtrLift.mmAs = pMold->ExtrLift.mmAs;
		if(0 == gMachineInfo.Calib)	/* 非调校模式  */
		{
			if(pMold->ExtrLift.Step > 0 && pMold->ExtrLift.Step < 20000)
			{
				pMold->ExtrLift.Step = 0;
				//	pMold->ExtrLift.Step = 40000; //ipis081
				pMold->Alarm.ExtrliftCalErr = 1;
			}
		}
		else if(0 == pMold->ExtrLift.NetworkInit)
		{
			if(pMold->ExtrLift.Step > 0 && pMold->ExtrLift.Step < 20000)
			{
				pMold->ExtrLift.Step = 0;
			}
		}
	}/* if(1 == pMold->ExtrLift.CalOK) */

	/*  toggle carriage linear  */
	pExtrLiftFix->ToggleLin[0].X = 0.0;
	pExtrLiftFix->ToggleLin[0].Y = 0.0;

	pExtrLiftFix->ToggleLin[ToggleLinNodeNum-1].X = pExtrLiftFix->Length;
	pExtrLiftFix->ToggleLin[ToggleLinNodeNum-1].Y = pExtrLiftFix->Length;

	TogLinearR.Y = pMold->ExtrLift.mmAsDrive;
	HydLinear(&TogLinearR);

	if(TogLinearR.status != 0)
	{
		pMold->Alarm.ExtrliftLinNotOK = 1;
		pMold->ExtrLift.mmAs = pMold->ExtrLift.mmAsDrive;
	}
	else
	{
		pMold->ExtrLift.mmAs = TogLinearR.X;
	}

	/* network and calibration is ok, axis has an error   */
	if(0 == pMold->ExtrLift.AxisReady)
	{
		if(pMold->ExtrLift.Step > 0 && pMold->ExtrLift.Step < 20000)
		{
			pMold->ExtrLift.Step = 30000;
		}
	}

	/*  relative position  */
	pMold->ExtrLift.Ss = pMold->ExtrLift.As;
	pMold->ExtrLift.mmAsMax = pExtrLiftFix->Length + 10;

	/* gAlarm time value    */
	if(!pMold->TimeSet.ExtrLiftUpAlarmTime)pMold->TimeSet.ExtrLiftUpAlarmTime = 1000;   /* 10s  */
	if(!pMold->TimeSet.ExtrLiftDnAlarmTime)pMold->TimeSet.ExtrLiftDnAlarmTime = 1000;   /* 10s  */

	/* Up or down  position flag  */
	if(1 == pMold->ExtrLift.CalOK)
	{
		pMold->ExtrLift.UpPos = pMold->TransDIn.ExtruderLiftUpLimit
			&& (pMold->ExtrLift.mmAs > (pExtrLiftPara->S_Up - pMold->ExtrLift.Tolerance))
			&& (pMold->ExtrLift.mmAs < (pExtrLiftPara->S_Up + pMold->ExtrLift.Tolerance));

		pMold->ExtrLift.DnPos = pMold->TransDIn.ExtruderLiftDnLimit
			&& (pMold->ExtrLift.mmAs < (pExtrLiftPara->S_Dn + pMold->ExtrLift.Tolerance))
			&& (pMold->ExtrLift.mmAs > (pExtrLiftPara->S_Dn - pMold->ExtrLift.Tolerance));

	}
	else
	{
		pMold->ExtrLift.UpPos = 0;
		pMold->ExtrLift.DnPos = 0;
	}

	/* ------------------ current position ------------------ */
	pMold->ExtrLift.vProfGen.s_act = pMold->ExtrLift.mmAsDrive;
	pMold->ExtrLift.vProfGen.v_act = pMold->ExtrLift.v_act;

	/* Up or down move step */
	switch (pMold->ExtrLift.Step )
	{
		/*------------------ stop all the Output ------------------*/
		case 0:

			pMold->ActInfo.ExtrLiftUp  = 0;
			pMold->ActInfo.ExtrLiftDn  = 0;

			pMold->ExtrLift.p_set = 0;
			pMold->ExtrLift.v_set = 0;

			pMold->ExtrLift.Timer.IN = 0;
			pMold->ExtrLift.LimitTimer.IN = 0;
			break;

		/*------------------ Extrlift up -------------------- */
		case 100: /* up delay*/
			if(pMold->Option.ExtrLift)
			{
				if(pMold->TimeSet.ExtrLiftUpDelay != 0)
				{
					pMold->ExtrLift.Timer.IN = 1;
					pMold->ExtrLift.Timer.PT = pMold->TimeSet.ExtrLiftUpDelay;
					pMold->ExtrLift.Step 	= 200;
				}
				else
				{
					pMold->ExtrLift.Step = 300;
				}
			}
			else
			{
				pMold->ExtrLift.Step = 2900;
			}
			break;

		case 200: /*delay ok*/
			pMold->TimeDis.ExtrLiftUpDelay = pMold->ExtrLift.Timer.ET;
			if (1 == pMold->ExtrLift.Timer.Q)
			{
				pMold->ExtrLift.Timer.IN     = 0;
				//	pMold->TimeDis.ExtrLiftUpDelay = 0;
				pMold->ExtrLift.Step = 300;
			}
			break;

		case 300:
			if(0 == pMold->ExtrLift.UpHWSwitch)
			{

				/* xTogLinearLTrans */
				pMold->ExtrLift.S_UpDrive = xTogLinearRTrans(pExtrLiftPara->S_Up);

				pMold->ExtrLift.LimitTimer.IN = 1;
				pMold->ExtrLift.LimitTimer.PT = pMold->TimeSet.ExtrLiftUpAlarmTime;

				pMold->ExtrLift.vProfGen.Ts = tTask;
				pMold->ExtrLift.vProfGen.Tj = pExtrLiftFix->Up.Tj;
				pMold->ExtrLift.vProfGen.Td = pExtrLiftFix->Up.Td;

				pMold->ExtrLift.vProfGen.accel = pExtrLiftFix->Up.accel;
				if(pMold->ExtrLift.vProfGen.accel <= 0.0)pMold->ExtrLift.vProfGen.accel = 1000;

				pMold->ExtrLift.vProfGen.decel = pExtrLiftFix->Up.accel;
				if(pMold->ExtrLift.vProfGen.decel <= 0.0)pMold->ExtrLift.vProfGen.decel = 1000;

				pMold->ExtrLift.vProfGen.decel_end = pExtrLiftFix->Up.decel_end;
				if(pMold->ExtrLift.vProfGen.decel_end <= 0.0)pMold->ExtrLift.vProfGen.decel_end = 100;

				pMold->ExtrLift.vProfGen.v_start = 0;
				pMold->ExtrLift.vProfGen.v_end = 0.0;
				pMold->ExtrLift.vProfGen.s_end = pMold->ExtrLift.S_UpDrive;
				pMold->ExtrLift.vProfGen.init = 1;

				pMold->ExtrLift.Step = 400;
			}
			else
			{
				pMold->HwAlarm.ExtrLiftUpHWSwitch = 1;
				pMold->ExtrLift.Step = 40000;
			}
			break;

		case 400:	/* up */
			pMold->ActInfo.ExtrLiftUp  = 1;

			pMold->ExtrLift.vProfGen.v_set = pMold->ExtrLift.V_Up;
			HydvProfGen(&pMold->ExtrLift.vProfGen);

			pMold->ExtrLift.p_set = pExtrLiftPara->P_Up = 100.0;
			pMold->ExtrLift.v_set = pMold->ExtrLift.vProfGen.v_out;

			pMold->ExtrLift.actTjUp = pMold->ExtrLift.vProfGen.Tj;

			pMold->TimeDis.ExtrLiftUpAlarmTime = pMold->ExtrLift.LimitTimer.ET;

			if(pMold->ExtrLift.vProfGen.s_act >= pMold->ExtrLift.vProfGen.s_end - pExtrLiftFix->Tolerance)
			{
				pMold->ExtrLift.LimitTimer.IN = 0;
				pMold->ExtrLift.p_set = 0;
				pMold->ExtrLift.v_set = 0;
				pMold->ExtrLift.Step = 500;
			}
			if(1 == pMold->ExtrLift.UpHWSwitch)
			{
				pMold->HwAlarm.ExtrLiftUpHWSwitch = 1;
				pMold->ExtrLift.Step = 40000;
			}
			break;

		case 500:
			pMold->ActInfo.ExtrLiftUp = 0;
			pMold->ExtrLift.p_set = 0;
			pMold->ExtrLift.v_set = 0;

			if (1==gMachineInfo.Auto)
			{
				pMold->ExtrLift.Step = 10100;
			}
			else
			{
				pMold->ExtrLift.Step = 2900;
			}

			break;

		case 2900:
			pMold->ActInfo.ExtrLiftUp = 0;
			pMold->ActInfo.ExtrLiftDn = 0;

			pMold->ExtrLift.p_set = 0;
			pMold->ExtrLift.v_set = 0;

			pMold->ExtrLift.Timer.IN    = 0;
			pMold->ExtrLift.LimitTimer.IN = 0;

			pMold->ExtrLift.Step = 3000;
			break;

		case 3000:
			break;

		/*  --------------- Calibration Extrlift up --------------- */
		case 5000:
			if(0 == pMold->ExtrLift.UpHWSwitch)
			{
				pMold->ActInfo.ExtrLiftUp  = 1;

				pMold->ExtrLift.p_set = pExtrLiftFix->pCalibMax;
				pMold->ExtrLift.v_set = pExtrLiftFix->vCalibMax;

			}
			if(1 == pMold->ExtrLift.UpHWSwitch)
			{
				pMold->HwAlarm.ExtrLiftUpHWSwitch = 1;
				pMold->ExtrLift.Step = 40000;
			}
			break;

		/*--------------- Extrlift down -----------------*/
		case 10100: /* down delay*/
			if (pMold->TimeSet.ExtrLiftDnDelay != 0)
			{
				pMold->ExtrLift.Timer.IN = 1;
				pMold->ExtrLift.Timer.PT = pMold->TimeSet.ExtrLiftDnDelay;
				pMold->ExtrLift.Step = 10200;
			}
			else
			{
				pMold->ExtrLift.Step = 10300;
			}
			break;

		case 10200: /*delay ok*/
			pMold->TimeDis.ExtrLiftDnDelay = pMold->ExtrLift.Timer.ET;
			if (1 == pMold->ExtrLift.Timer.Q)
			{
				pMold->ExtrLift.Timer.IN = 0;
				//	pMold->TimeDis.ExtrLiftDnDelay = 0;
				pMold->ExtrLift.Step = 10300;
			}
			break;

		case 10300:
			if(0 == pMold->ExtrLift.DnHWSwitch)
			{
				/* xTogLinearLTrans */
				pMold->ExtrLift.S_DnDrive = xTogLinearRTrans(pExtrLiftPara->S_Dn);

				pMold->ExtrLift.LimitTimer.IN = 1;
				pMold->ExtrLift.LimitTimer.PT = pMold->TimeSet.ExtrLiftDnAlarmTime;

				pMold->ExtrLift.vProfGen.Ts = tTask;
				pMold->ExtrLift.vProfGen.Tj = pExtrLiftFix->Dn.Tj;
				pMold->ExtrLift.vProfGen.Td = pExtrLiftFix->Dn.Td;

				pMold->ExtrLift.vProfGen.accel = pExtrLiftFix->Dn.accel;
				if(pMold->ExtrLift.vProfGen.accel <= 0.0)pMold->ExtrLift.vProfGen.accel = 1000;

				pMold->ExtrLift.vProfGen.decel = pExtrLiftFix->Dn.accel;
				if(pMold->ExtrLift.vProfGen.decel <= 0.0)pMold->ExtrLift.vProfGen.decel = 1000;

				pMold->ExtrLift.vProfGen.decel_end = pExtrLiftFix->Dn.decel_end;
				if(pMold->ExtrLift.vProfGen.decel_end <= 0.0)pMold->ExtrLift.vProfGen.decel_end = 100;

				pMold->ExtrLift.vProfGen.v_start = 0;
				pMold->ExtrLift.vProfGen.v_end = 0.0;
				pMold->ExtrLift.vProfGen.s_end = pMold->ExtrLift.S_DnDrive;
				pMold->ExtrLift.vProfGen.init = 1;

				pMold->ExtrLift.Step = 10400;
			}
			else
			{
				pMold->HwAlarm.ExtrLiftDnHWSwitch = 1;
				pMold->ExtrLift.Step = 40000;
			}
			break;

		case 10400:	/* down */
			pMold->ActInfo.ExtrLiftDn  = 1;

			pMold->ExtrLift.vProfGen.v_set = pMold->ExtrLift.V_Dn;
			HydvProfGen(&pMold->ExtrLift.vProfGen);

			pMold->ExtrLift.p_set = pExtrLiftPara->P_Dn = 100.0;
			pMold->ExtrLift.v_set = pMold->ExtrLift.vProfGen.v_out;

			pMold->ExtrLift.actTjDn = pMold->ExtrLift.vProfGen.Tj;

			pMold->TimeDis.ExtrLiftDnAlarmTime = pMold->ExtrLift.LimitTimer.ET;

			if(pMold->ExtrLift.vProfGen.s_act <= pMold->ExtrLift.vProfGen.s_end + pExtrLiftFix->Tolerance)
			{
				pMold->ExtrLift.LimitTimer.IN = 0;
				pMold->ExtrLift.v_set = 0;
				pMold->ExtrLift.p_set = 0;
				pMold->ExtrLift.Step = 10500;
			}
			if(1 == pMold->ExtrLift.DnHWSwitch)
			{
				pMold->HwAlarm.ExtrLiftDnHWSwitch = 1;
				pMold->ExtrLift.Step = 40000;
			}
			break;

		case 10500:
			pMold->ActInfo.ExtrLiftUp = 0;
			pMold->ActInfo.ExtrLiftDn = 0;

			pMold->ExtrLift.p_set = 0;
			pMold->ExtrLift.v_set = 0;

			pMold->ExtrLift.Timer.IN    = 0;
			pMold->ExtrLift.LimitTimer.IN = 0;

			pMold->ExtrLift.Step = 13000;
			break;

		case 13000:
			break;

		/*  --------------- Calibration Extrlift down --------------- */
		case 15000:
			if(0 == pMold->ExtrLift.DnHWSwitch)
			{
				pMold->ActInfo.ExtrLiftDn  = 1;

				pMold->ExtrLift.p_set = pExtrLiftFix->pCalibMax;
				pMold->ExtrLift.v_set = -pExtrLiftFix->vCalibZero;

			}
			if(1 == pMold->ExtrLift.DnHWSwitch)
			{
				pMold->HwAlarm.ExtrLiftDnHWSwitch = 1;
				pMold->ExtrLift.Step = 40000;
			}
			break;

		/* ----------------------------  manual stop ------------------------- */
		case 20000:
			pMold->ExtrLift.Timer.IN      = 0;
			pMold->ExtrLift.LimitTimer.IN = 0;

			pMold->ActInfo.ExtrLiftUp = 0;
			pMold->ActInfo.ExtrLiftDn = 0;

			pMold->ExtrLift.p_old = pMold->ExtrLift.p_set;

			pMold->ExtrLift.Step = 21000;
			break;

		case 21000:
			pMold->ExtrLift.vRamp.Internal.Once = 0;
			pMold->ExtrLift.vRamp.Set = pMold->ExtrLift.v_set;

			pMold->ExtrLift.vRamp.Ts = tTask;

			if(pMold->ExtrLift.v_set > 0)
			{
				pMold->ExtrLift.vRamp.Accel = pExtrLiftFix->Dn.accel_stop;
			}
			else
			{
				pMold->ExtrLift.vRamp.Accel = pExtrLiftFix->Up.accel_stop;
			}

			/* call profile function */
			HydSCurveRamp(&pMold->ExtrLift.vRamp);

			pMold->ExtrLift.p_set = pMold->ExtrLift.p_old;
			pMold->ExtrLift.v_set = pMold->ExtrLift.vRamp.Out;

			pMold->ExtrLift.Step = 22000;
			break;

		case 22000:
			pMold->ExtrLift.vRamp.Ts = tTask;
			pMold->ExtrLift.vRamp.Set = 0.0;

			/* call profile function */
			HydSCurveRamp(&pMold->ExtrLift.vRamp);

			pMold->ExtrLift.p_set = pMold->ExtrLift.p_old;
			pMold->ExtrLift.v_set = pMold->ExtrLift.vRamp.Out;

			if(pMold->ExtrLift.v_set < 0.1 && pMold->ExtrLift.v_set > -0.1)
			{
				pMold->ExtrLift.v_set = 0.0;
				pMold->ExtrLift.Step = 0;
			}
			break;

		/* ----------------------------  Instance stop ------------------------- */
		case 30000:
			pMold->ExtrLift.Timer.IN      = 0;
			pMold->ExtrLift.LimitTimer.IN = 0;

			pMold->ActInfo.ExtrLiftUp = 0;
			pMold->ActInfo.ExtrLiftDn = 0;

			pMold->ExtrLift.vRamp.Internal.Once = 0;
			pMold->ExtrLift.vRamp.Set = pMold->ExtrLift.v_set;

			pMold->ExtrLift.vRamp.Ts = tTask;

			pMold->ExtrLift.vRamp.Accel = INSTANCY_STOP_DECEL;
			HydSCurveRamp(&pMold->ExtrLift.vRamp);

			pMold->ExtrLift.p_set = 100.0;
			pMold->ExtrLift.v_set = pMold->ExtrLift.vRamp.Out;

			pMold->ExtrLift.Step = 31000;
			break;

		case 31000:
			pMold->ExtrLift.vRamp.Ts = tTask;
			pMold->ExtrLift.vRamp.Set = 0.0;

			HydSCurveRamp(&pMold->ExtrLift.vRamp);

			pMold->ExtrLift.p_set = 100.0;
			pMold->ExtrLift.v_set = pMold->ExtrLift.vRamp.Out;

			if(pMold->ExtrLift.v_set < 0.1 && pMold->ExtrLift.v_set > -0.1)
			{
				pMold->ExtrLift.v_set = 0.0;
				pMold->ExtrLift.Step  = 0;
			}
			break;

		/* ----------------------------  Error step ------------------------- */
		case 40000:
			pMold->ExtrLift.Timer.IN      = 0;
			pMold->ExtrLift.LimitTimer.IN = 0;

			pMold->ActInfo.ExtrLiftUp = 0;
			pMold->ActInfo.ExtrLiftDn = 0;

			pMold->ExtrLift.v_set = 0.0;
			break;

		/* ----------------------------  auto run stop ------------------------- */
		case 41000:
			pMold->ExtrLift.Timer.IN      = 0;
			pMold->ExtrLift.LimitTimer.IN = 0;

			pMold->ActInfo.ExtrLiftUp = 0;
			pMold->ActInfo.ExtrLiftDn = 0;

			pMold->ExtrLift.Step = 42000;
			break;

		case 42000:
			pMold->ExtrLift.vRamp.Internal.Once = 0;
			pMold->ExtrLift.vRamp.Set = pMold->ExtrLift.v_set;

			pMold->ExtrLift.vRamp.Ts = tTask;

			pMold->ExtrLift.vRamp.Accel = INSTANCY_STOP_DECEL;

			/* call profile function */
			HydSCurveRamp(&pMold->ExtrLift.vRamp);
			pMold->ExtrLift.Step = 43000;
			break;

		case 43000:
			pMold->ExtrLift.vRamp.Ts = tTask;
			pMold->ExtrLift.vRamp.Set = 0.0;

			/* call profile function */
			HydSCurveRamp(&pMold->ExtrLift.vRamp);

			pMold->ExtrLift.p_set = 100.0;
			pMold->ExtrLift.v_set = pMold->ExtrLift.vRamp.Out;

			if(pMold->ExtrLift.v_set < 0.1 && pMold->ExtrLift.v_set > -0.1)
			{
				pMold->ExtrLift.v_set = 0.0;
				pMold->ExtrLift.Step = 40000;
			}
			break;
	}/* end of switch */

	/* ----------------- ExtrLift Up / down timeout --------------------  */
	if(1 == pMold->ExtrLift.LimitTimer.Q && 1 == gMachineInfo.TimeLimit)
	{
		if(pMold->ExtrLift.Step < 500 && pMold->ExtrLift.Step > 200)		/* ExtrLift Up  */
		{
			pMold->Alarm.ExtrLiftNotAtUpPos = 1;
		}

		if(pMold->ExtrLift.Step < 10500 && pMold->ExtrLift.Step > 10200)		/* ExtrLift Dn  */
		{
			pMold->Alarm.ExtrLiftNotAtDnPos = 1;
		}

		pMold->ExtrLift.LimitTimer.IN = 0;
		pMold->ExtrLift.Step = 40000;

		if(gMachineInfo.Auto)
		{
			gMachineInfo.ExtrliftAlarmReqSemiAutoFlag = 1;
		}
	}
}
REAL xTogLinearRTrans(REAL pTogLinPos)
{
	xTogLinearR.Y = pTogLinPos;
	HydLinear(&xTogLinearR);
	if(0 == xTogLinearR.status)
	{
		return xTogLinearR.X;
	}
	else
	{
		return 0;
	}
}
```

#### extrlift.var
```iecst
VAR
	cntTime : UDINT;
	tTask : REAL := 0.0;
	RTInfo_Task : RTInfo := (0);
	tErrorDelay : REAL;
	vActHydDT2_R : HydDT2;
	vActHydDT2_L : HydDT2;
END_VAR
(*Toggle*)
VAR
	ToggleROld : ARRAY[0..30] OF Hyd_Node_typ;
	TogLinearR : HydLinear;
	xToggleNodeR : ARRAY[0..30] OF Hyd_Node_typ;
	xTogLinearR : HydLinear;
	oldToggleLinNodeNum : USINT;
	ToggleLinNodeNum : USINT;
	bToggle_Init : USINT;
END_VAR
```

### Program Logical/process/lowblow (ANSIC, version 1.00.0) - Low pressure blowing

#### lowblow.c
```c
/********************************************************************
 * COPYRIGHT --  B&R China
 ********************************************************************
 * Program: LowBlow
 * File: LowBlow.c
 * Author: lijianjun
 * Created: March 06, 2013
 ********************************************************************
 * Implementation of program LowBlow --- 1 blowing
 ********************************************************************/

#include <bur/plctypes.h>

#ifdef _DEFAULT_INCLUDES
	#include <AsDefault.h>
#endif

/**************************************************************************************
                            Function Declarations
**************************************************************************************/

void BlowCBM( Mold_typ * pMold);
void BlowStandard( Mold_typ * pMold);

/**************************************************************************************
     	        		I N I T U P  O F   T H E   T A S K
**************************************************************************************/
_INIT void init ( void )
 {
 		LMold.LowBlow.Step = 0;
 		RMold.LowBlow.Step = 0;
 } /* end of _INIT */

 /*************************************************************************************
        				C Y C L I C   P A R T   O F   T H E   T A S K
**************************************************************************************/

 _CYCLIC void cyclic ( void )
 {
	if(1 == gMachineFix.Option.bBlowModeCBM)
	{
		BlowCBM(&LMold);
		BlowCBM(&RMold);
	}
	else
	{
		BlowStandard(&LMold);
		BlowStandard(&RMold);
	}

//	gMachineOut.LMold.LowBlow = LMold.LowBlow.Out;
//	gMachineOut.RMold.LowBlow = RMold.LowBlow.Out;
} /* end of _CYCLIC */

void BlowCBM( Mold_typ * pMold)
{
	switch ( pMold->LowBlow.Step )
	{
		/*------------------ stop all the output ------------------*/
		case 0:
			pMold->LowBlow.Out  		= 0;
			pMold->ActInfo.LowBlow   = 0;
			pMold->LowBlow.Timer.IN	= 0;
			break;

		/*------------------ Blow  -------------------- */
		case 100: /* blow delay*/
			pMold->LowBlow.TimerTotal.IN = 0;
			if(pMold->TimeSet.LowBlowDelay != 0)
			{
				pMold->LowBlow.Timer.IN = 1;
				pMold->LowBlow.Timer.PT = pMold->TimeSet.LowBlowDelay;
				pMold->LowBlow.Step 	   = 200;
			}
			else
			{
				pMold->LowBlow.Step = 300;
			}
			break;

		case 200: /* delay ok */
			pMold->TimeDis.LowBlowDelay = pMold->LowBlow.Timer.ET;
			if (1 == pMold->LowBlow.Timer.Q)
			{
				pMold->LowBlow.Timer.IN     = 0;
			//	pMold->TimeDis.LowBlowDelay = 0;

				pMold->LowBlow.Step = 300;
			}
			break;

		case 300:
			pMold->LowBlow.TimerTotal.IN = 1;
			pMold->LowBlow.TimerTotal.PT = pMold->TimeSet.TotalBlowTime * 10;

			if(pMold->HighBlow.Step > 300)
			{
				pMold->HighBlow.Step = 470;
			}

			if(pMold->TimeSet.LowBlowTime != 0)
			{
				pMold->LowBlow.Timer.IN = 1;
				pMold->LowBlow.Timer.PT = pMold->TimeSet.LowBlowTime;
				pMold->LowBlow.Step = 400;
			}
			else
			{
				pMold->LowBlow.Step = 450;
			}
			break;

		case 400:	/* pre blow time   */
			pMold->LowBlow.Out     = 1;
			pMold->ActInfo.LowBlow = 1;
			pMold->TimeDis.LowBlowTime = pMold->LowBlow.Timer.ET;
			if (1 == pMold->LowBlow.Timer.Q)
			{
				pMold->LowBlow.Out      = 0;
				pMold->LowBlow.Timer.IN = 0;
			//	pMold->TimeDis.LowBlowTime = 0;
				pMold->LowBlow.Step = 450;
			}

			if (1 == pMold->LowBlow.TimerTotal.Q || 1 == pMold->HighBlow.TimerTotal.Q)
			{
				pMold->LowBlow.Out = 0;
				pMold->LowBlow.TimerTotal.IN = 0;

				pMold->LowBlow.Step = 480;
			}
			break;

		case 450:
			pMold->LowBlow.Out     = 1;
			pMold->ActInfo.LowBlow = 1;

			if (1 == pMold->LowBlow.TimerTotal.Q || 1 == pMold->HighBlow.TimerTotal.Q)
			{
				pMold->LowBlow.Out = 0;
				pMold->LowBlow.TimerTotal.IN = 0;
				pMold->LowBlow.Step = 480;
			}
			break;

		case 470:
			pMold->LowBlow.Out = 0;
			break;

		case 480:
			if(pMold->HighBlow.Step < 480 && pMold->HighBlow.Step > 0)pMold->HighBlow.Step = 480;
			pMold->LowBlow.Out      = 0;
			pMold->LowBlow.Timer.IN = 0;
			pMold->LowBlow.TimerTotal.IN = 0;
			pMold->LowBlow.Step = 900;
			break;

		case 900:
			pMold->LowBlow.Out      = 0;
			pMold->LowBlow.Timer.IN = 0;

//			pMold->TimeDis.LowBlowTime  = 0;
//			pMold->TimeDis.LowBlowDelay = 0;

			pMold->ActInfo.LowBlow = 0;

			pMold->LowBlow.Step = 3000;
			break;

		case 3000:
			break;

		case 5000:
			pMold->LowBlow.Out     = 1;
			pMold->ActInfo.LowBlow = 1;
			break;

		case 20000:
			pMold->LowBlow.Out      = 0;
			pMold->LowBlow.Timer.IN = 0;
			pMold->LowBlow.TimerTotal.IN = 0;

//			pMold->TimeDis.LowBlowTime  = 0;
//			pMold->TimeDis.LowBlowDelay = 0;

			pMold->ActInfo.LowBlow= 0;
			pMold->LowBlow.Step 	 = 0;
			break;

		case 30000:
			pMold->LowBlow.Out      = 0;
			pMold->LowBlow.Timer.IN = 0;
			pMold->LowBlow.TimerTotal.IN = 0;

//			pMold->TimeDis.LowBlowTime  = 0;
//			pMold->TimeDis.LowBlowDelay = 0;

			pMold->ActInfo.LowBlow  = 0;
			pMold->LowBlow.Step     = 0;
			break;

	}/* end of switch */
}/*end of function */

void BlowStandard( Mold_typ * pMold)
{
	switch ( pMold->LowBlow.Step )
	{
		/*------------------ stop all the output ------------------*/
		case 0:
			pMold->LowBlow.Out  		= 0;
			pMold->ActInfo.LowBlow   = 0;
			pMold->LowBlow.Timer.IN	= 0;
			break;

		/*------------------ Blow  -------------------- */
		case 100: /* blow delay*/
			pMold->LowBlow.TimerTotal.IN = 0;
			if(pMold->TimeSet.LowBlowDelay != 0)
			{
				pMold->LowBlow.Timer.IN = 1;
				pMold->LowBlow.Timer.PT = pMold->TimeSet.LowBlowDelay;
				pMold->LowBlow.Step 	   = 200;
			}
			else
			{
				pMold->LowBlow.Step = 300;
			}
			break;

		case 200: /* delay ok */
			pMold->TimeDis.LowBlowDelay = pMold->LowBlow.Timer.ET;
			if (1 == pMold->LowBlow.Timer.Q)
			{
				pMold->LowBlow.Timer.IN     = 0;
		//		pMold->TimeDis.LowBlowDelay = 0;

				pMold->LowBlow.Step = 300;
			}
			break;

		case 300:
			if(pMold->TimeSet.LowBlowTime != 0)
			{
				pMold->LowBlow.Timer.IN = 1;
				pMold->LowBlow.Timer.PT = pMold->TimeSet.LowBlowTime;
				pMold->LowBlow.Step = 400;
			}
			else
			{
				pMold->LowBlow.Step = 900;
			}
			break;

		case 400:	/* pre blow time   */
			pMold->LowBlow.Out     = 1;
			pMold->ActInfo.LowBlow = 1;
			pMold->TimeDis.LowBlowTime = pMold->LowBlow.Timer.ET;
			if (1 == pMold->LowBlow.Timer.Q)
			{
				pMold->LowBlow.Out      = 0;
				pMold->LowBlow.Timer.IN = 0;
			//	pMold->TimeDis.LowBlowTime = 0;
				pMold->LowBlow.Step = 900;
			}
			break;

		case 900:
			pMold->LowBlow.Out      = 0;
			pMold->LowBlow.Timer.IN = 0;

//			pMold->TimeDis.LowBlowTime  = 0;
//			pMold->TimeDis.LowBlowDelay = 0;

			pMold->ActInfo.LowBlow = 0;

			pMold->LowBlow.Step = 3000;
			break;

		case 3000:
			break;

		case 20000:
			pMold->LowBlow.Out      = 0;
			pMold->LowBlow.Timer.IN = 0;
			pMold->LowBlow.TimerTotal.IN = 0;

//			pMold->TimeDis.LowBlowTime  = 0;
//			pMold->TimeDis.LowBlowDelay = 0;

			pMold->ActInfo.LowBlow= 0;
			pMold->LowBlow.Step 	 = 0;
			break;

		case 30000:
			pMold->LowBlow.Out      = 0;
			pMold->LowBlow.Timer.IN = 0;
			pMold->LowBlow.TimerTotal.IN = 0;

//			pMold->TimeDis.LowBlowTime  = 0;
//			pMold->TimeDis.LowBlowDelay = 0;

			pMold->ActInfo.LowBlow  = 0;
			pMold->LowBlow.Step     = 0;
			break;

	}/* end of switch */
}/*end of function */
```

### Program Logical/process/highblow (ANSIC, version 1.00.0) - Main blowing air

#### highblow.c
```c
/********************************************************************
 * COPYRIGHT --  B&R China
 ********************************************************************
 * Program: HighBlow
 * File: HighBlow.c
 * Author: lijianjun
 * Created: March 06, 2013
 ********************************************************************
 * Implementation of program HighBlow --- 2 blowing
 ********************************************************************/

#include <bur/plctypes.h>

#ifdef _DEFAULT_INCLUDES
	#include <AsDefault.h>
#endif

/**************************************************************************************
                            Function Declarations
**************************************************************************************/

void BlowCBM( Mold_typ * pMold);
void BlowStandard( Mold_typ * pMold);
void BlowStandardNew( Mold_typ * pMold, Option_Fix_typ * pOptionFix);
void BlowFreezing( Mold_typ * pMold);
/**************************************************************************************
     	        		I N I T U P  O F   T H E   T A S K
**************************************************************************************/
_INIT void init ( void )
 {
 	LMold.HighBlow.Step = 0;
 	RMold.HighBlow.Step = 0;
 } /* end of _INIT */

 /*************************************************************************************
        				C Y C L I C   P A R T   O F   T H E   T A S K
**************************************************************************************/

 _CYCLIC void cyclic ( void )
 {
	bHideBlowStandard = gMachineFix.Option.bBlowModeCBM;
	bHideBlowCBM      = !gMachineFix.Option.bBlowModeCBM;

	bHideLowBlow = !gMachineFix.Option.bLowBlow;

	if(0 == gPanelObj.LevelBand_4 && 0 == bHideLowBlow)
	{
		bHideLowBlowIO = 0;
	}
	else
	{
		bHideLowBlowIO = 1;
	}
	gMachineFix.Option.bBlowModeCBM =0; //ipis0802
	if(1 == gMachineFix.Option.bBlowModeCBM)
	{
		BlowCBM(&LMold);
		BlowCBM(&RMold);
	}
	else
	{
//		BlowStandard(&LMold);
//		BlowStandard(&RMold);

		switch (gMachineFix.MoldR.Blow.eBlowMode)
		{
			case BLOW_MODE_STANDARD:

				BlowStandardNew(&RMold,&gMachineFix.Option);
				BlowStandardNew(&LMold,&gMachineFix.Option);

				break;

			case BLOW_MODE_FREEZINGBLOW:

				BlowFreezing(&RMold);
				BlowFreezing(&LMold);
				break;
		}
	}

//	switch(LMold.HighBlow.Out)
//	{
//		case 0:		/* 关闭  */
//			gMachineOut.LMold.HighBlow = 0;
//			gMachineOut.LMold.Exhaust = 0;
//
//			break;
//
//		case 2:		/* 高壓吹氣 -- 循环吹起  */
//			gMachineOut.LMold.HighBlow  = 1;
//			gMachineOut.LMold.Exhaust = 0;
//			break;
//
//		case 3:		/* 循环放气  */
//			gMachineOut.LMold.HighBlow  = 0;
//			gMachineOut.LMold.Exhaust = 1;
//			break;
//
//		case 4:		/* 高壓吹風延时  */
//			gMachineOut.LMold.HighBlow  = 0;
//			gMachineOut.LMold.Exhaust = 0;
//			break;
//
//		case 5:		/* 放气  */
//			gMachineOut.LMold.HighBlow  = 0;
//			gMachineOut.LMold.Exhaust = 1;
//			break;
//
//		case 6:
//			gMachineOut.LMold.HighBlow  = 1;
//			gMachineOut.RMold.Exhaust = 0;
//			break;
//	}/* switch(LMold.HighBlow.Out) */
//
//	switch(RMold.HighBlow.Out)
//	{
//		case 0:		/* 关闭  */
//			gMachineOut.RMold.HighBlow = 0;
//			gMachineOut.RMold.Exhaust = 0;
//
//			break;
//
//		case 2:		/* 高壓吹風 -- 循环吹風  */
//			gMachineOut.RMold.HighBlow = 1;
//			gMachineOut.RMold.Exhaust  = 0;
//			break;
//
//		case 3:		/* 循环放風  */
//			gMachineOut.RMold.HighBlow = 0;
//			gMachineOut.RMold.Exhaust  = 1;
//			break;
//
//		case 4:		/* 高壓吹風延时  */
//			gMachineOut.RMold.HighBlow  = 0;
//			gMachineOut.RMold.Exhaust = 0;
//			break;
//
//		case 5:		/* 放气  */
//			gMachineOut.RMold.HighBlow  = 0;
//			gMachineOut.RMold.Exhaust = 1;
//			break;
//
//		case 6:
//			gMachineOut.RMold.HighBlow  = 1;
//			gMachineOut.RMold.Exhaust = 0;
//			break;
//
//	}/* switch(RMold.HighBlow.Out) */
//
//	gMachineOut.LMold.ExhaustForBlow2 =LMold.ValveOut.ExhaustForBlow2;
//	gMachineOut.RMold.ExhaustForBlow2 = RMold.ValveOut.ExhaustForBlow2;

//	gMachineOut.LMold.HighBlow =  LMold.HighBlow.Out;
//	gMachineOut.RMold.HighBlow =  RMold.HighBlow.Out;

	gMachineOut.RMold.HighBlow =  RMold.ValveOut.HighBlow;
	gMachineOut.LMold.HighBlow =  LMold.ValveOut.HighBlow;

	gMachineOut.RMold.LowBlow =  RMold.ValveOut.LowBlow;
	gMachineOut.LMold.LowBlow =  LMold.ValveOut.LowBlow;

	gMachineOut.RMold.FreezingBlow =  RMold.ValveOut.FreezingBlow;
	gMachineOut.LMold.FreezingBlow =  LMold.ValveOut.FreezingBlow;

	gMachineOut.RMold.Exhaust =  RMold.ValveOut.Exhaust;
	gMachineOut.LMold.Exhaust =  LMold.ValveOut.Exhaust;

	/*------------- BlowMode--------------- */
	gMachineFix.MoldL.Blow.eBlowMode = gMachineFix.MoldR.Blow.eBlowMode;

 } /* end of _CYCLIC */

void BlowCBM( Mold_typ * pMold)
{
	if(pMold->TimeSet.TotalBlowTime * 10 < pMold->TimeSet.BlowingTime)
	{
		pMold->TimeSet.TotalBlowTime = pMold->TimeSet.BlowingTime/10;
	}

	if(pMold->HighBlow.TimerTotal.ET > pMold->LowBlow.TimerTotal.ET)
	{
		pMold->TimeDis.TotalBlowTime = pMold->HighBlow.TimerTotal.ET/10;
	}
	else
	{
		pMold->TimeDis.TotalBlowTime = pMold->LowBlow.TimerTotal.ET/10;
	}

	switch ( pMold->HighBlow.Step )
	{
		/*------------------ stop all the output ------------------*/
		case 0:
			pMold->HighBlow.Out  		= 0;
			pMold->ActInfo.HighBlow   = 0;
			pMold->HighBlow.Timer.IN	= 0;
			break;

		/*------------------ Blow  -------------------- */
		case 100:
			pMold->HighBlow.TimerTotal.IN = 0;
			if(pMold->TimeSet.BlowingDelay != 0)
			{
				pMold->HighBlow.Timer.IN = 1;
				pMold->HighBlow.Timer.PT = pMold->TimeSet.BlowingDelay;
				pMold->HighBlow.Step 	   = 200;
			}
			else
			{
			//	pMold->HighBlow.Step = 300;
			pMold->HighBlow.Step = 700;
			}
			break;

		case 200: /* high blowing delay ok */
			pMold->HighBlow.Out = 4;
			pMold->ActInfo.HighBlow = 1;
			pMold->TimeDis.BlowingDelay = pMold->HighBlow.Timer.ET;
			if (1 == pMold->HighBlow.Timer.Q)
			{
				pMold->HighBlow.Timer.IN      = 0;
			//	pMold->TimeDis.BlowingDelay = 0;

				pMold->HighBlow.Step = 300;  //ipis
		//	pMold->HighBlow.Step = 700;   // ipis
			}
			break;

		case 300:
			pMold->HighBlow.TimerTotal.IN = 1;
			pMold->HighBlow.TimerTotal.PT = pMold->TimeSet.TotalBlowTime * 10;

			if(pMold->LowBlow.Step > 300)
			{
				pMold->LowBlow.Step = 470;
			}

			if(pMold->TimeSet.BlowingTime != 0)
			{
				pMold->HighBlow.tCounter = 0;
				pMold->HighBlow.Timer.IN = 1;
				pMold->HighBlow.Timer.PT = pMold->TimeSet.BlowingTime;
				pMold->HighBlow.Step = 400;

			}
			else
			{
				pMold->HighBlow.Step = 450;
			}
			break;

		case 400:	/* high blowing time   */
			pMold->HighBlow.Out     = 2;
			pMold->ActInfo.HighBlow = 1;
			pMold->TimeDis.BlowingTime = pMold->HighBlow.Timer.ET;
			if (1 == pMold->HighBlow.Timer.Q)
			{
				pMold->HighBlow.Timer.IN = 0;
			//	pMold->TimeDis.BlowingTime = 0;
				pMold->HighBlow.Step = 450; /* 900; */
			}

			if (1 == pMold->LowBlow.TimerTotal.Q || 1 == pMold->HighBlow.TimerTotal.Q)
			{
				pMold->HighBlow.Out = 0;
				pMold->HighBlow.TimerTotal.IN = 0;

				pMold->HighBlow.Step = 480;
			}
			break;

		case 450:
			pMold->HighBlow.Out     = 2;
			pMold->ActInfo.HighBlow = 1;

			if (1 == pMold->LowBlow.TimerTotal.Q || 1 == pMold->HighBlow.TimerTotal.Q)
			{
				pMold->HighBlow.Out = 0;
				pMold->HighBlow.TimerTotal.IN = 0;
				pMold->HighBlow.Step = 480;
			}
			break;

		case 470:
			pMold->HighBlow.Out = 0;
			break;

		case 480:
			if(pMold->LowBlow.Step < 480 && pMold->LowBlow.Step > 0)pMold->LowBlow.Step = 480;
			pMold->HighBlow.Out = 0;
			pMold->HighBlow.Timer.IN = 0;
			pMold->HighBlow.TimerTotal.IN = 0;
			pMold->HighBlow.Step = 1100;
			break;

		case 500:
			if((pMold->TimeSet.TotalBlowTime * 10 - pMold->TimeSet.BlowingTime) > 0)
			{
				pMold->HighBlow.tCounter = 0;
				pMold->HighBlow.Timer.IN = 1;
				pMold->HighBlow.Timer.PT = pMold->TimeSet.TotalBlowTime * 10 - pMold->TimeSet.BlowingTime;
				pMold->HighBlow.Step = 600;
			}
			else
			{
				pMold->HighBlow.Out  = 0;
				pMold->HighBlow.Step = 1100;
			}
			break;

		case 600:
			pMold->HighBlow.tCounter++;

			if(pMold->Option.IntervalBlow)
			{
				if((0 == pMold->TimeSet.InterValBlowOnTime) || (0 == pMold->TimeSet.InterValBlowOffTime))
				{
					pMold->HighBlow.Out     = 2;
					pMold->ActInfo.HighBlow = 1;
				}
				else
				{
					pMold->HighBlow.tTemp = pMold->HighBlow.tCounter % (pMold->TimeSet.InterValBlowOnTime + pMold->TimeSet.InterValBlowOffTime);
					if(pMold->HighBlow.tTemp <= pMold->TimeSet.InterValBlowOnTime)
					{
						pMold->HighBlow.Out     = 2;
						pMold->ActInfo.HighBlow = 1;
						pMold->TimeDis.InterValBlowOnTime  = pMold->HighBlow.tTemp;
					//	pMold->TimeDis.InterValBlowOffTime = 0;
					}
					else
					{
						pMold->HighBlow.Out     = 3;
						pMold->ActInfo.HighBlow = 0;
					//	pMold->TimeDis.InterValBlowOnTime = 0;
						pMold->TimeDis.InterValBlowOffTime = pMold->HighBlow.tTemp - pMold->TimeSet.InterValBlowOnTime;
					}
				}
			}/* if(pMold->Option.InterValBlow) */
			else
			{
				pMold->HighBlow.Out     = 2;
				pMold->ActInfo.HighBlow = 1;
			}

			pMold->TimeDis.TotalBlowTime = (pMold->HighBlow.Timer.ET + pMold->TimeSet.BlowingTime)/10;
			if (1 == pMold->HighBlow.Timer.Q)
			{
				pMold->HighBlow.Out      = 0;
				pMold->HighBlow.Timer.IN = 0;
//				pMold->TimeDis.TotalBlowTime       = 0;
//				pMold->TimeDis.InterValBlowOnTime  = 0;
//				pMold->TimeDis.InterValBlowOffTime = 0;

				pMold->HighBlow.Step = 1100;
			}
			break;

		/*--------------------------------------------------------------------------------------*/

//		case 700:
//			if(pMold->TimeSet.BlowingTime != 0)
//			{
//				pMold->HighBlow.tCounter = 0;
//				pMold->HighBlow.Timer.IN = 1;
//				pMold->HighBlow.Timer.PT = pMold->TimeSet.BlowingTime;
//				pMold->HighBlow.Step = 710;
//			}
//			else
//			{
//				pMold->HighBlow.Step = 720;
//			}
//
//		break;
//
//		case 710:/* high blowing time   */
//			pMold->HighBlow.Out     = 2;
//			pMold->ActInfo.HighBlow = 1;
//			pMold->TimeDis.BlowingTime = pMold->HighBlow.Timer.ET;
//			if (1 == pMold->HighBlow.Timer.Q)
//			{
//				pMold->HighBlow.Timer.IN = 0;
//				//	pMold->TimeDis.BlowingTime = 0;
//				pMold->HighBlow.Step = 720;
//			}
//
//		break;
//
//		case 720: /*AirVentingTime*/
//
//			if(pMold->TimeSet.AirVentingTime != 0)
//			{
//
//				pMold->HighBlow.Timer.IN = 1;
//				pMold->HighBlow.Timer.PT = pMold->TimeSet.AirVentingTime;
//				pMold->HighBlow.Step = 730;
//			}
//			else
//			{
//				pMold->HighBlow.Step = 760;
//			}
//		break;
//
//		case 730:/* AirVentingTime   */
//			pMold->HighBlow.Out     = 3;
//			pMold->ActInfo.HighBlow = 0;
//			pMold->TimeDis.AirVentingTime = pMold->HighBlow.Timer.ET;
//			if (1 == pMold->HighBlow.Timer.Q)
//			{
//				pMold->HighBlow.Timer.IN = 0;
//				//	pMold->TimeDis.AirVentingTime = 0;
//				pMold->HighBlow.Step = 760;
//			}
//
//			break;
//
//
//		case 760: /* high blowing time2   */
//			if(pMold->TimeSet.BlowingTime2 != 0)
//			{
//				pMold->HighBlow.tCounter = 0;
//				pMold->HighBlow.Timer.IN = 1;
//				pMold->HighBlow.Timer.PT = pMold->TimeSet.BlowingTime2;
//				pMold->HighBlow.Step = 770;
//			}
//			else
//			{
//				pMold->HighBlow.Step = 780;
//			}
//
//			break;
//
//		case 770:/* high blowing time2   */
//			pMold->HighBlow.Out     = 2;
//			pMold->ActInfo.HighBlow = 1;
//			pMold->TimeDis.BlowingTime2 = pMold->HighBlow.Timer.ET;
//			if (1 == pMold->HighBlow.Timer.Q)
//			{
//				pMold->HighBlow.Timer.IN = 0;
//				//	pMold->TimeDis.BlowingTime2 = 0;
//				pMold->HighBlow.Step = 780;
//			}
//
//			break;
//
//		case 780: /*AirVentingTime2*/
//
//			if(pMold->TimeSet.AirVentingTime2 != 0)
//			{
//
//				pMold->HighBlow.Timer.IN = 1;
//				pMold->HighBlow.Timer.PT = pMold->TimeSet.AirVentingTime2;
//				pMold->HighBlow.Step = 790;
//			}
//			else
//			{
//				pMold->HighBlow.Step = 1300;
//			}
//			break;
//
//		case 790:/* AirVentingTime2  */
//			pMold->HighBlow.Out     = 3;
//			pMold->ActInfo.HighBlow = 0;
//			pMold->TimeDis.AirVentingTime2 = pMold->HighBlow.Timer.ET;
//			if (1 == pMold->HighBlow.Timer.Q)
//			{
//				pMold->HighBlow.Timer.IN = 0;
//				//	pMold->TimeDis.AirVentingTime2 = 0;
//				pMold->HighBlow.Step = 1300;
//			}
//
//			break;

		case 1100:
			if(1 == gMachineInfo.Auto)
			{
//				pMold->PullBottom.Step  = 100; 		/*  拉底启动  */

				/*if(pMold->BlowPin.Step < 500 && pMold->BlowPin.Step > 100)pMold->BlowPin.Step = 500;  blow pin down force end  */

				pMold->LowBlow.Step = 900;				/*  低壓吹風強制結束 */
			}

			pMold->ActInfo.HighBlow = 0;

			if(pMold->TimeSet.AirVentingTime != 0)
			{
				pMold->HighBlow.Timer.IN = 1;
				pMold->HighBlow.Timer.PT = pMold->TimeSet.AirVentingTime;	/*  排气时间  */

				pMold->HighBlow.Step = 1200;
			}
			else
			{
				pMold->HighBlow.Step = 1300;
			}
			break;

		case 1200:
			pMold->HighBlow.Out = 5;
			pMold->TimeDis.AirVentingTime = pMold->HighBlow.Timer.ET;
			if (1 == pMold->HighBlow.Timer.Q)
			{
				pMold->HighBlow.Timer.IN = 0;
			//	pMold->TimeDis.AirVentingTime = 0;
				pMold->HighBlow.Step = 1300;
			}
			break;

		case 1300:
			pMold->HighBlow.Out      = 0;
			pMold->HighBlow.Timer.IN = 0;

//			pMold->TimeDis.BlowingDelay   = 0;
//			pMold->TimeDis.BlowingTime    = 0;
//			pMold->TimeDis.AirVentingTime = 0;

			pMold->ActInfo.HighBlow  = 0;

			pMold->Lock.Step  = 10100;	/*  卸压 */
			pMold->HighBlow.Step = 3000;
			break;
		case 3000:
			break;

		case 5000:
			pMold->HighBlow.Out = 6;
			break;

		case 20000:
			pMold->HighBlow.Out      = 0;
			pMold->HighBlow.Timer.IN = 0;
			pMold->HighBlow.TimerTotal.IN = 0;

//			pMold->TimeDis.InterValBlowOnTime  = 0;
//			pMold->TimeDis.InterValBlowOffTime = 0;
//
//			pMold->TimeDis.BlowingDelay   = 0;
//			pMold->TimeDis.BlowingTime    = 0;
//
//			pMold->TimeDis.TotalBlowTime  = 0;
//			pMold->TimeDis.AirVentingTime = 0;

			pMold->ActInfo.HighBlow= 0;
			pMold->HighBlow.Step 	 = 0;
			break;

		case 30000:
			pMold->HighBlow.Out      = 0;
			pMold->HighBlow.Timer.IN = 0;
			pMold->HighBlow.TimerTotal.IN = 0;

//			pMold->TimeDis.InterValBlowOnTime  = 0;
//			pMold->TimeDis.InterValBlowOffTime = 0;
//
//			pMold->TimeDis.BlowingDelay   = 0;
//			pMold->TimeDis.BlowingTime    = 0;
//
//			pMold->TimeDis.TotalBlowTime  = 0;
//			pMold->TimeDis.AirVentingTime = 0;

			pMold->ActInfo.HighBlow  = 0;
			pMold->HighBlow.Step     = 0;
			break;

	}/* end of switch */
}/*end of function */

void BlowStandard( Mold_typ * pMold)
{
	if(pMold->TimeSet.TotalBlowTime * 10 < pMold->TimeSet.BlowingTime)
	{
		pMold->TimeSet.TotalBlowTime = pMold->TimeSet.BlowingTime/10;
	}

	pMold->TimeDis.TotalBlowTime = pMold->HighBlow.TimerTotal.ET/10;

	switch ( pMold->HighBlow.Step )
	{
		/*------------------ stop all the output ------------------*/
		case 0:
			pMold->HighBlow.Out  		= 0;
			pMold->ActInfo.HighBlow   = 0;
			pMold->HighBlow.Timer.IN	= 0;
			break;

		/*------------------ Blow  -------------------- */
		case 100:
			pMold->HighBlow.TimerTotal.IN = 0;
			if(pMold->TimeSet.BlowingDelay != 0)
			{
				pMold->HighBlow.Timer.IN = 1;
				pMold->HighBlow.Timer.PT = pMold->TimeSet.BlowingDelay;
				pMold->HighBlow.Step 	   = 200;

				//gExSPC
				if(pMold == & LMold)
				{
					gExSPC[ExIndex].LMold.BlowingDelay = pMold->TimeSet.BlowingDelay/100.0;
				}
				else
				{
					gExSPC[ExIndex].RMold.BlowingDelay = pMold->TimeSet.BlowingDelay/100.0;
				}

			}
			else
			{
				pMold->HighBlow.Step = 700;
			}
			break;

		case 200: /* high blowing delay ok */
			pMold->HighBlow.Out = 4;
			pMold->ActInfo.HighBlow = 1;
			pMold->TimeDis.BlowingDelay = pMold->HighBlow.Timer.ET;
			if (1 == pMold->HighBlow.Timer.Q)
			{
				pMold->HighBlow.Timer.IN      = 0;
		//		pMold->TimeDis.BlowingDelay = 0;

			//	pMold->HighBlow.Step = 300;
				pMold->HighBlow.Step = 700;
			}
			break;

		case 300:

			pMold->HighBlow.Out = 4;
			pMold->ActInfo.HighBlow = 1;
			pMold->HighBlow.TimerTotal.IN = 1;
			pMold->HighBlow.TimerTotal.PT = pMold->TimeSet.TotalBlowTime * 10;

			if(pMold->TimeSet.BlowingTime != 0)
			{
				pMold->HighBlow.tCounter = 0;
				pMold->HighBlow.Timer.IN = 1;
				pMold->HighBlow.Timer.PT = pMold->TimeSet.BlowingTime;
				pMold->HighBlow.Step = 400;
			}
			else
			{
				pMold->HighBlow.Step = 500;
			}
			break;

		case 400:	/* high blowing time   */
			pMold->HighBlow.Out     = 2;
			pMold->ActInfo.HighBlow = 1;
			pMold->TimeDis.BlowingTime = pMold->HighBlow.Timer.ET;
			if (1 == pMold->HighBlow.Timer.Q)
			{
				pMold->HighBlow.Timer.IN = 0;
			//	pMold->TimeDis.BlowingTime = 0;
				pMold->HighBlow.Step = 500;
			}

			if (1 == pMold->HighBlow.TimerTotal.Q)
			{
				pMold->HighBlow.Out = 0;
				pMold->HighBlow.TimerTotal.IN = 0;

				pMold->HighBlow.Step = 1100;
			}
			break;

		case 500:
			if((pMold->TimeSet.TotalBlowTime * 10 - pMold->TimeSet.BlowingTime) > 0)
			{
				pMold->HighBlow.tCounter = 0;
				pMold->HighBlow.Timer.IN = 1;
				pMold->HighBlow.Timer.PT = pMold->TimeSet.TotalBlowTime * 10 - pMold->TimeSet.BlowingTime;
				pMold->HighBlow.Step = 600;
			}
			else
			{
				pMold->HighBlow.Out  = 0;
				pMold->HighBlow.Step = 1100;
			}
			break;

		case 600:
			pMold->HighBlow.tCounter++;

			if(pMold->Option.IntervalBlow)
			{
				if((0 == pMold->TimeSet.InterValBlowOnTime) || (0 == pMold->TimeSet.InterValBlowOffTime))
				{
					pMold->HighBlow.Out     = 2;
					pMold->ActInfo.HighBlow = 1;
				}
				else
				{
					pMold->HighBlow.tTemp = pMold->HighBlow.tCounter % (pMold->TimeSet.InterValBlowOnTime + pMold->TimeSet.InterValBlowOffTime);
					if(pMold->HighBlow.tTemp <= pMold->TimeSet.InterValBlowOnTime)
					{
						pMold->HighBlow.Out     = 2;
						pMold->ActInfo.HighBlow = 1;
						pMold->TimeDis.InterValBlowOnTime  = pMold->HighBlow.tTemp;
					//	pMold->TimeDis.InterValBlowOffTime = 0;
					}
					else
					{
						pMold->HighBlow.Out     = 3;
						pMold->ActInfo.HighBlow = 0;
					//	pMold->TimeDis.InterValBlowOnTime = 0;
						pMold->TimeDis.InterValBlowOffTime = pMold->HighBlow.tTemp - pMold->TimeSet.InterValBlowOnTime;
					}
				}
			}/* if(pMold->Option.InterValBlow) */
			else
			{
				pMold->HighBlow.Out     = 2;
				pMold->ActInfo.HighBlow = 1;
			}

			pMold->TimeDis.TotalBlowTime = (pMold->HighBlow.Timer.ET + pMold->TimeSet.BlowingTime)/10;
			if (1 == pMold->HighBlow.Timer.Q)
			{
				pMold->HighBlow.Out      = 0;
				pMold->HighBlow.Timer.IN = 0;
//				pMold->TimeDis.TotalBlowTime       = 0;
//				pMold->TimeDis.InterValBlowOnTime  = 0;
//				pMold->TimeDis.InterValBlowOffTime = 0;

				pMold->HighBlow.Step = 1100;
			}
			break;

		/*--------------------------------------------------------------------------------------*/

		case 700:
			if(pMold->TimeSet.BlowingTime != 0)
			{
				pMold->HighBlow.tCounter = 0;
				pMold->HighBlow.Timer.IN = 1;
				pMold->HighBlow.Timer.PT = pMold->TimeSet.BlowingTime;
				pMold->HighBlow.Step = 710;

				//gExSPC
				if(pMold == & LMold)
				{
					gExSPC[ExIndex].LMold.BlowingTime = pMold->TimeSet.BlowingTime/100.0;
				}
				else
				{
					gExSPC[ExIndex].RMold.BlowingTime = pMold->TimeSet.BlowingTime/100.0;
				}
			}
			else
			{
				pMold->HighBlow.Step = 720;
			}

			break;

		case 710:/* high blowing time   */
			pMold->HighBlow.Out     = 2;
			pMold->ActInfo.HighBlow = 1;
			pMold->TimeDis.BlowingTime = pMold->HighBlow.Timer.ET;
			if (1 == pMold->HighBlow.Timer.Q)
			{
				pMold->HighBlow.Timer.IN = 0;
				//	pMold->TimeDis.BlowingTime = 0;
				pMold->HighBlow.Step = 720;
			}

			break;

		case 720: /*AirVentingTime*/

			if(pMold->TimeSet.AirVentingTime != 0)
			{

				pMold->HighBlow.Timer.IN = 1;
				pMold->HighBlow.Timer.PT = pMold->TimeSet.AirVentingTime;
				pMold->HighBlow.Step = 730;

				//gExSPC
				if(pMold == & LMold)
				{
					gExSPC[ExIndex].LMold.AirVentingTime = pMold->TimeSet.AirVentingTime/100.0;
				}
				else
				{
					gExSPC[ExIndex].RMold.AirVentingTime = pMold->TimeSet.AirVentingTime/100.0;
				}
			}
			else
			{
				pMold->HighBlow.Step = 760;
			}
			break;

		case 730:/* AirVentingTime   */
			pMold->HighBlow.Out     = 3;
			pMold->ActInfo.HighBlow = 0;
			pMold->TimeDis.AirVentingTime = pMold->HighBlow.Timer.ET;
			if (1 == pMold->HighBlow.Timer.Q)
			{
				pMold->HighBlow.Timer.IN = 0;
				//	pMold->TimeDis.AirVentingTime = 0;
				pMold->HighBlow.Step = 760;
			}

			break;

		case 760: /* high blowing time2   */
			if(pMold->TimeSet.BlowingTime2 != 0)
			{
				pMold->HighBlow.tCounter = 0;
				pMold->HighBlow.Timer.IN = 1;
				pMold->HighBlow.Timer.PT = pMold->TimeSet.BlowingTime2;
				pMold->HighBlow.Step = 770;

				//gExSPC
				if(pMold == & LMold)
				{
					gExSPC[ExIndex].LMold.BlowingTime2 = pMold->TimeSet.BlowingTime2/100.0;
				}
				else
				{
					gExSPC[ExIndex].RMold.BlowingTime2 = pMold->TimeSet.BlowingTime2/100.0;
				}

			}
			else
			{
				pMold->HighBlow.Step = 780;
			}

			break;

		case 770:/* high blowing time2   */
			pMold->HighBlow.Out     = 2;
			pMold->ActInfo.HighBlow = 1;
			pMold->ValveOut.ExhaustForBlow2   = 1; //ipis0219
			pMold->TimeDis.BlowingTime2 = pMold->HighBlow.Timer.ET;
			if (1 == pMold->HighBlow.Timer.Q)
			{
				pMold->HighBlow.Timer.IN = 0;
		//s	pMold->ValveOut.ExhaustForBlow2   = 0; //ipis0219
				//	pMold->TimeDis.BlowingTime2 = 0;
				pMold->HighBlow.Step = 780;
			}

			break;

		case 780: /*AirVentingTime2*/

			if(pMold->TimeSet.AirVentingTime2 != 0)
			{

				pMold->HighBlow.Timer.IN = 1;
				pMold->HighBlow.Timer.PT = pMold->TimeSet.AirVentingTime2;
				pMold->HighBlow.Step = 790;

				//gExSPC
				if(pMold == & LMold)
				{
					gExSPC[ExIndex].LMold.AirVentingTime2 = pMold->TimeSet.AirVentingTime2/100.0;
				}
				else
				{
					gExSPC[ExIndex].RMold.AirVentingTime2 = pMold->TimeSet.AirVentingTime2/100.0;
				}
			}
			else
			{
				pMold->HighBlow.Step = 1300;
			}
			break;

		case 790:/* AirVentingTime2  */
			pMold->HighBlow.Out     = 3;
			pMold->ActInfo.HighBlow = 0;
			pMold->TimeDis.AirVentingTime2 = pMold->HighBlow.Timer.ET;
			if (1 == pMold->HighBlow.Timer.Q)
			{
				pMold->HighBlow.Timer.IN = 0;
				//	pMold->TimeDis.AirVentingTime2 = 0;
				pMold->HighBlow.Step = 1300;
			}

			break;

		case 1100:
			if(1 == gMachineInfo.Auto)
			{
				pMold->PullBottom.Step  = 100; 		/*  拉底启动  */

				/*if(pMold->BlowPin.Step < 500 && pMold->BlowPin.Step > 100)pMold->BlowPin.Step = 500;   blow pin down force end  */

				pMold->LowBlow.Step = 900;				/*  低壓吹風強制結束 */
			}

			pMold->ActInfo.HighBlow = 0;

			if(pMold->TimeSet.AirVentingTime != 0)
			{
				pMold->HighBlow.Timer.IN = 1;
				pMold->HighBlow.Timer.PT = pMold->TimeSet.AirVentingTime;	/*  排气时间  */

				pMold->HighBlow.Step = 1200;
			}
			else
			{
				pMold->HighBlow.Step = 1300;
			}
			break;

		case 1200:
			pMold->HighBlow.Out = 5;
			pMold->TimeDis.AirVentingTime = pMold->HighBlow.Timer.ET;
			if (1 == pMold->HighBlow.Timer.Q)
			{
				pMold->HighBlow.Timer.IN = 0;
		//		pMold->TimeDis.AirVentingTime = 0;
				pMold->HighBlow.Step = 1300;
			}
			break;

		case 1300:
			pMold->HighBlow.Out      = 0;
			pMold->HighBlow.Timer.IN = 0;
				pMold->ValveOut.ExhaustForBlow2   = 0; //ipis0219
//			pMold->TimeDis.BlowingDelay   = 0;
//			pMold->TimeDis.BlowingTime    = 0;
//			pMold->TimeDis.AirVentingTime = 0;

			pMold->ActInfo.HighBlow  = 0;

			pMold->Lock.Step  = 10100;	/*  卸压 */
			pMold->HighBlow.Step = 3000;
			break;
		case 3000:
			break;

		case 5000:
			pMold->HighBlow.Out = 6;
			break;

		case 20000:
			pMold->HighBlow.Out      = 0;
			pMold->HighBlow.Timer.IN = 0;
			pMold->HighBlow.TimerTotal.IN = 0;
			pMold->ValveOut.ExhaustForBlow2   = 0; //ipis0219
//			pMold->TimeDis.InterValBlowOnTime  = 0;
//			pMold->TimeDis.InterValBlowOffTime = 0;
//
//			pMold->TimeDis.BlowingDelay   = 0;
//			pMold->TimeDis.BlowingTime    = 0;
//
//			pMold->TimeDis.TotalBlowTime  = 0;
//			pMold->TimeDis.AirVentingTime = 0;

			pMold->ActInfo.HighBlow= 0;
			pMold->HighBlow.Step 	 = 0;
			break;

		case 30000:
			pMold->HighBlow.Out      = 0;
			pMold->HighBlow.Timer.IN = 0;
			pMold->HighBlow.TimerTotal.IN = 0;
				pMold->ValveOut.ExhaustForBlow2   = 0; //ipis0219
//			pMold->TimeDis.InterValBlowOnTime  = 0;
//			pMold->TimeDis.InterValBlowOffTime = 0;
//
//			pMold->TimeDis.BlowingDelay   = 0;
//			pMold->TimeDis.BlowingTime    = 0;
//
//			pMold->TimeDis.TotalBlowTime  = 0;
//			pMold->TimeDis.AirVentingTime = 0;

			pMold->ActInfo.HighBlow  = 0;
			pMold->HighBlow.Step     = 0;
			break;
	}/* end of switch */
}/*end of function */

void BlowStandardNew( Mold_typ * pMold, Option_Fix_typ * pOptionFix)
{

	switch ( pMold->HighBlow.Step )
	{
		/*------------------ stop all the output ------------------*/
		case 0:
			pMold->ActInfo.HighBlow   	= 0;
			pMold->ValveOut.HighBlow  	= 0;
			pMold->ValveOut.LowBlow 	= 0;

			pMold->HighBlow.Timer.IN	= 0;
			break;

		/*------------------ Blow  -------------------- */
		case 100:
			if(pMold->TimeSet.BlowingDelay != 0)
			{
				pMold->HighBlow.Timer.IN = 1;
				pMold->HighBlow.Timer.PT = pMold->TimeSet.BlowingDelay;
				pMold->HighBlow.Step 	   = 200;
			}
			else
			{
				pMold->HighBlow.Step = 210;
			}
			break;

		case 200: /* high blowing delay ok */
			pMold->TimeDis.BlowingDelay = pMold->HighBlow.Timer.ET;
			if (1 == pMold->HighBlow.Timer.Q)
			{
				pMold->HighBlow.Timer.IN = 0;
				pMold->HighBlow.Step = 210;
			}
			break;

		case 210: /*  pre Low blowing ok */
			if(pMold->TimeSet.PreBlowTime != 0)
			{
				pMold->HighBlow.Timer.IN = 1;
				pMold->HighBlow.Timer.PT = pMold->TimeSet.PreBlowTime;
				pMold->HighBlow.Step = 220;
			}
			else
			{
				pMold->HighBlow.Step = 300;
			}

			break;

		case 220:/* pre low blowing time   */
			pMold->ActInfo.HighBlow = 1;

			pMold->ValveOut.LowBlow = 1;
			pMold->TimeDis.PreBlowTime = pMold->HighBlow.Timer.ET;
			if (1 == pMold->HighBlow.Timer.Q)
			{
				pMold->ActInfo.HighBlow = 0;
				pMold->ValveOut.LowBlow = 0;
				pMold->HighBlow.Timer.IN = 0;
				//	pMold->TimeDis.PreBlowTime = 0;
				pMold->HighBlow.Step = 300;
			}

			break;

		case 300:
			if(pMold->TimeSet.BlowingTime != 0)
			{
				pMold->HighBlow.Timer.IN = 1;
				pMold->HighBlow.Timer.PT = pMold->TimeSet.BlowingTime;
				pMold->HighBlow.Step = 400;
			}
			else
			{
				pMold->HighBlow.Step = 500;
			}

			break;

		case 400:/* high blowing time   */
			pMold->ActInfo.HighBlow = 1;

			pMold->ValveOut.HighBlow = 1;
			pMold->TimeDis.BlowingTime = pMold->HighBlow.Timer.ET;
			if (1 == pMold->HighBlow.Timer.Q)
			{
				pMold->ActInfo.HighBlow  = 0;
				pMold->ValveOut.HighBlow = 0;
				pMold->HighBlow.Timer.IN = 0;
				//	pMold->TimeDis.BlowingTime = 0;
				pMold->HighBlow.Step = 500;
			}

			break;

		case 500: /*AirVentingTime Set*/
			if(pMold->TimeSet.AirVentingTime != 0)
			{
				pMold->HighBlow.Timer.IN = 1;
				pMold->HighBlow.Timer.PT = pMold->TimeSet.AirVentingTime;
				pMold->HighBlow.Step = 600;
			}
			else
			{
				pMold->HighBlow.Step = 700;
			}
			break;

		case 600:/* AirVentingTime   */
			pMold->ActInfo.HighBlow = 0;

			pMold->ValveOut.HighBlow = 0;
			pMold->ValveOut.LowBlow = 0;
			pMold->TimeDis.AirVentingTime = pMold->HighBlow.Timer.ET;
			if (1 == pMold->HighBlow.Timer.Q)
			{
				pMold->HighBlow.Timer.IN = 0;
				//	pMold->TimeDis.AirVentingTime = 0;
				pMold->HighBlow.Step = 700;
			}

			break;

		case 700: /* high blowing time2 Set  */
			if(pMold->TimeSet.BlowingTime2 != 0)
			{
				pMold->HighBlow.Timer.IN = 1;
				pMold->HighBlow.Timer.PT = pMold->TimeSet.BlowingTime2;
				pMold->HighBlow.Step = 800;
			}
			else
			{
				pMold->HighBlow.Step = 900;
			}

			break;

		case 800:/* high blowing time2   */
			pMold->ActInfo.HighBlow = 1;

			if( 0 == pOptionFix->bBlowingTime2LowBlow)
			{
				pMold->ValveOut.HighBlow = 1;
			}
			else
			{
				pMold->ValveOut.LowBlow = 1;
			}

			pMold->TimeDis.BlowingTime2 = pMold->HighBlow.Timer.ET;
			if (1 == pMold->HighBlow.Timer.Q)
			{
				pMold->ActInfo.HighBlow  = 0;
				pMold->ValveOut.HighBlow = 0;
				pMold->ValveOut.LowBlow  = 0;
				pMold->HighBlow.Timer.IN = 0;
				//	pMold->TimeDis.BlowingTime2 = 0;
				pMold->HighBlow.Step = 900;
			}

			break;

		case 900: /*AirVentingTime2 Set*/

			if(pMold->TimeSet.AirVentingTime2 != 0)
			{
				pMold->HighBlow.Timer.IN = 1;
				pMold->HighBlow.Timer.PT = pMold->TimeSet.AirVentingTime2;
				pMold->HighBlow.Step = 1000;
			}
			else
			{
				pMold->HighBlow.Step = 1300;
			}
			break;

		case 1000:/* AirVentingTime2  */
			pMold->ValveOut.HighBlow = 0;
			pMold->ValveOut.LowBlow = 0;
			pMold->ActInfo.HighBlow = 0;
			pMold->TimeDis.AirVentingTime2 = pMold->HighBlow.Timer.ET;
			if (1 == pMold->HighBlow.Timer.Q)
			{
				pMold->HighBlow.Timer.IN = 0;
				//	pMold->TimeDis.AirVentingTime2 = 0;
				pMold->HighBlow.Step = 1300;
			}
			break;

		case 1300:
			pMold->ActInfo.HighBlow  = 0;

			pMold->ValveOut.HighBlow = 0;
			pMold->HighBlow.Timer.IN = 0;

			pMold->HighBlow.Step = 3000;
			break;

		case 3000:
			break;

		case 5000:
			pMold->ValveOut.HighBlow = 1;

			break;

		case 20000:
			pMold->ActInfo.HighBlow  = 0;

			pMold->ValveOut.HighBlow = 0;
			pMold->HighBlow.Timer.IN = 0;

			pMold->HighBlow.Step     = 0;
			break;

		case 30000:
			pMold->ActInfo.HighBlow  = 0;

			pMold->ValveOut.HighBlow = 0;
			pMold->HighBlow.Timer.IN = 0;

			pMold->HighBlow.Step     = 0;
			break;
	}/* end of switch */
}/*end of function */

void BlowFreezing( Mold_typ * pMold)
{

	switch ( pMold->HighBlow.Step )
	{
		/*------------------ stop all the output ------------------*/
		case 0:
			pMold->ActInfo.HighBlow  = 0;

			pMold->ValveOut.HighBlow = 0;
			pMold->ValveOut.FreezingBlow = 0;
			pMold->ValveOut.Exhaust = 0;
			pMold->HighBlow.Timer.IN = 0;
			break;

		/*------------------ Blow  -------------------- */
		case 100:
			if(pMold->TimeSet.BlowingDelay != 0)
			{
				pMold->HighBlow.Timer.IN = 1;
				pMold->HighBlow.Timer.PT = pMold->TimeSet.BlowingDelay;
				pMold->HighBlow.Step 	   = 200;
			}
			else
			{
				pMold->HighBlow.Step = 300;
			}
			break;

		case 200: /* high blowing delay ok */
			pMold->TimeDis.BlowingDelay = pMold->HighBlow.Timer.ET;
			if (1 == pMold->HighBlow.Timer.Q)
			{
				pMold->HighBlow.Timer.IN = 0;
				pMold->HighBlow.Step = 300;
			}
			break;

		case 300:
			if(pMold->TimeSet.BlowingTime != 0)
			{
				pMold->HighBlow.Timer.IN = 1;
				pMold->HighBlow.Timer.PT = pMold->TimeSet.BlowingTime;
				pMold->HighBlow.Step = 400;
			}
			else
			{
				pMold->HighBlow.Step = 500;
			}

			break;

		case 400:/* high blowing time   */
			pMold->ActInfo.HighBlow = 1;

			pMold->ValveOut.HighBlow = 1;
			pMold->TimeDis.BlowingTime = pMold->HighBlow.Timer.ET;
			if (1 == pMold->HighBlow.Timer.Q)
			{
				pMold->ActInfo.HighBlow  = 0;
				pMold->ValveOut.HighBlow = 0;
				pMold->HighBlow.Timer.IN = 0;
				//	pMold->TimeDis.BlowingTime = 0;
				pMold->HighBlow.Step = 500;
			}

			break;

		case 500: /*AirVentingTime Set*/
			if(pMold->TimeSet.AirVentingTime != 0)
			{
				pMold->HighBlow.Timer.IN = 1;
				pMold->HighBlow.Timer.PT = pMold->TimeSet.AirVentingTime;
				pMold->HighBlow.Step = 600;
			}
			else
			{
				pMold->HighBlow.Step = 700;
			}
			break;

		case 600:/* AirVentingTime   */
			pMold->ActInfo.HighBlow = 0;

			pMold->ValveOut.HighBlow = 0;
			pMold->ValveOut.Exhaust  = 1;
			pMold->TimeDis.AirVentingTime = pMold->HighBlow.Timer.ET;
			if (1 == pMold->HighBlow.Timer.Q)
			{
				pMold->ValveOut.Exhaust  = 0;
				pMold->HighBlow.Timer.IN = 0;
				//	pMold->TimeDis.AirVentingTime = 0;
				pMold->HighBlow.Step = 700;
			}

			break;

		case 700: /* high blowing time2 Set  */

			pMold->ValveOut.Exhaust  = 0;

			if(pMold->TimeSet.BlowingTime2 != 0)
			{
				pMold->HighBlow.Timer.IN = 1;
				pMold->HighBlow.Timer.PT = pMold->TimeSet.BlowingTime2;
				pMold->HighBlow.Step = 800;
			}
			else
			{
				pMold->HighBlow.Step = 900;
			}

			break;

		case 800:/* high blowing time2   */
			pMold->ActInfo.HighBlow = 1;

			pMold->ValveOut.FreezingBlow = 1;
			pMold->TimeDis.BlowingTime2 = pMold->HighBlow.Timer.ET;
			if (1 == pMold->HighBlow.Timer.Q)
			{
				pMold->ActInfo.HighBlow = 0;
				pMold->ValveOut.FreezingBlow = 0;
				pMold->HighBlow.Timer.IN = 0;
				//	pMold->TimeDis.BlowingTime2 = 0;
				pMold->HighBlow.Step = 900;
			}

			break;

		case 900: /*AirVentingTime2 Set*/
			pMold->ValveOut.FreezingBlow = 0;
			if(pMold->TimeSet.AirVentingTime2 != 0)
			{
				pMold->HighBlow.Timer.IN = 1;
				pMold->HighBlow.Timer.PT = pMold->TimeSet.AirVentingTime2;
				pMold->HighBlow.Step = 1000;
			}
			else
			{
				pMold->HighBlow.Step = 1300;
			}
			break;

		case 1000:/* AirVentingTime2  */
			pMold->ActInfo.HighBlow = 0;
			pMold->ValveOut.Exhaust = 1;
			pMold->TimeDis.AirVentingTime2 = pMold->HighBlow.Timer.ET;
			if (1 == pMold->HighBlow.Timer.Q)
			{
				pMold->HighBlow.Timer.IN = 0;
				//	pMold->TimeDis.AirVentingTime2 = 0;
				pMold->HighBlow.Step = 1300;
			}
			break;

		case 1300:
			pMold->ActInfo.HighBlow  = 0;

			pMold->ValveOut.HighBlow = 0;
			pMold->ValveOut.FreezingBlow = 0;
			pMold->ValveOut.Exhaust = 0;
			pMold->HighBlow.Timer.IN = 0;

			pMold->HighBlow.Step = 3000;
			break;

		case 3000:
			break;

		case 5000:
			pMold->ValveOut.HighBlow = 1;

			break;

		case 20000:
			pMold->ActInfo.HighBlow  = 0;

			pMold->ValveOut.HighBlow = 0;
			pMold->ValveOut.FreezingBlow = 0;
			pMold->ValveOut.Exhaust = 0;
			pMold->HighBlow.Timer.IN = 0;

			pMold->HighBlow.Step     = 0;
			break;

		case 30000:
			pMold->ActInfo.HighBlow  = 0;

			pMold->ValveOut.HighBlow = 0;
			pMold->ValveOut.FreezingBlow = 0;
			pMold->ValveOut.Exhaust = 0;
			pMold->HighBlow.Timer.IN = 0;

			pMold->HighBlow.Step     = 0;
			break;
	}/* end of switch */
}/*end of function */
```

#### highblow.var
```iecst
VAR
	bHideLowBlowIO : USINT;
	bHideLowBlow : USINT;
	bHideBlowCBM : USINT;
	bHideBlowStandard : USINT;
END_VAR
```

### Program Logical/process/bdeflash (ANSIC, version 1.00.0) - bottom deflash
